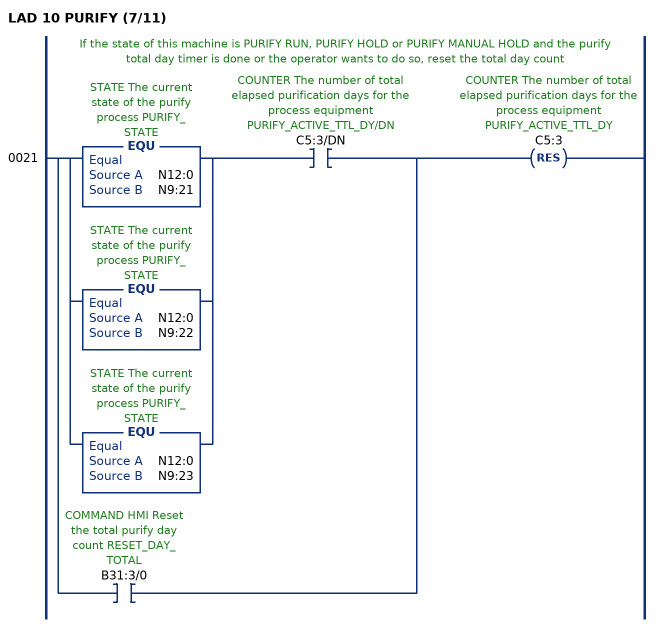
% Rung: 21 %
% If the state of this machine is PURIFY RUN, PURIFY HOLD or PURIFY MANUAL HOLD and the purify total day timer is done or the operator wants to do so, reset the total day count %
SOR BST BST EQU N12:0 N9:21 NXB EQU N12:0 N9:22 NXB EQU N12:0 N9:23 BND XIC C5:3/DN NXB XIC B31:3/0 BND RES C5:3 EOR
%   N12:0  PURIFY_STATE  "STATE The current state of the purify process" %
%   N9:21  PURIFY_RUN  "STATE Purify running" %
%   N9:22  PURIFY_HOLD  "STATE Purify Hold" %
%   N9:23  PURIFY_MANUAL_HOLD  "STATE Purify Manual Hold" %
%   C5:3  PURIFY_ACTIVE_TTL_DY  "COUNTER The number of total elapsed purification days for the process equipment" %
%   B31:3/0  RESET_DAY_TOTAL  "COMMAND HMI Reset the total purify day count" %

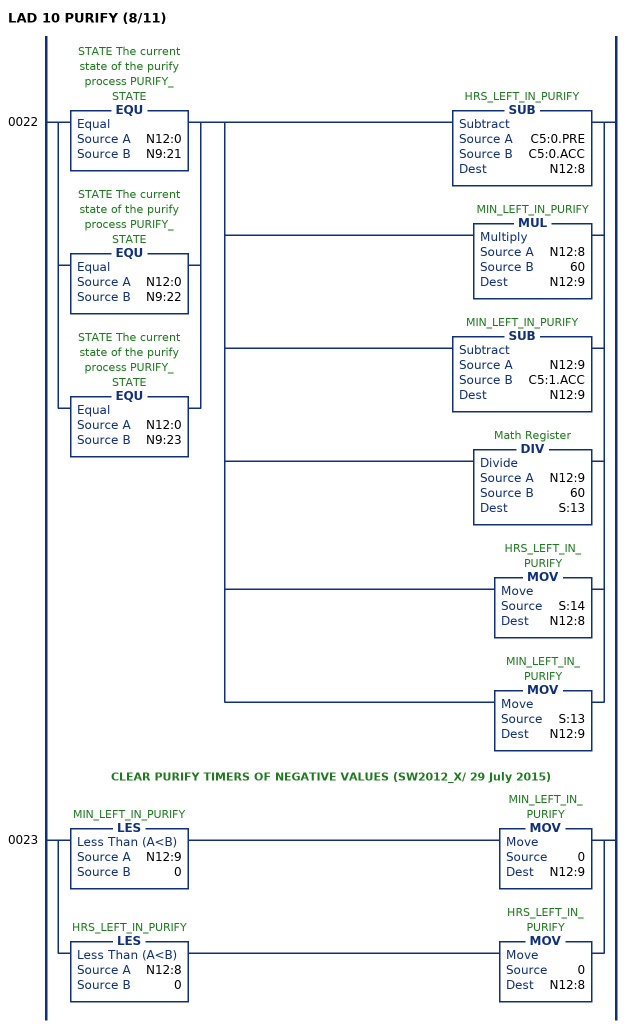
% Rung: 22 %
SOR BST EQU N12:0 N9:21 NXB EQU N12:0 N9:22 NXB EQU N12:0 N9:23 BND BST SUB C5:0.PRE C5:0.ACC N12:8 NXB MUL N12:8 60 N12:9 NXB SUB N12:9 C5:1.ACC N12:9 NXB DIV N12:9 60 S:13 NXB MOV S:14 N12:8 NXB MOV S:13 N12:9 BND EOR
%   N12:0  PURIFY_STATE  "STATE The current state of the purify process" %
%   N9:21  PURIFY_RUN  "STATE Purify running" %
%   N9:22  PURIFY_HOLD  "STATE Purify Hold" %
%   N9:23  PURIFY_MANUAL_HOLD  "STATE Purify Manual Hold" %
%   C5:0  PURIFY_ACTIVE_HOURS  "COUNTER The number of elapsed purification hours for the current ADS" %
%   N12:8  HRS_LEFT_IN_PURIFY %
%   N12:9  MIN_LEFT_IN_PURIFY %
%   C5:1  PURIFY_ACTIVE_MINUTE  "COUNTER The number of elapsed purification minutes for the current ADS (60 min)" %
%   S:13  "Math Register" %
%   S:14  "Math Register" %
% Rung: 23 %
% TITLE: CLEAR PURIFY TIMERS OF NEGATIVE VALUES (SW2012_X/ 29 July 2015) %
SOR BST LES N12:9 0 MOV 0 N12:9 NXB LES N12:8 0 MOV 0 N12:8 BND EOR
%   N12:9  MIN_LEFT_IN_PURIFY %
%   N12:8  HRS_LEFT_IN_PURIFY %

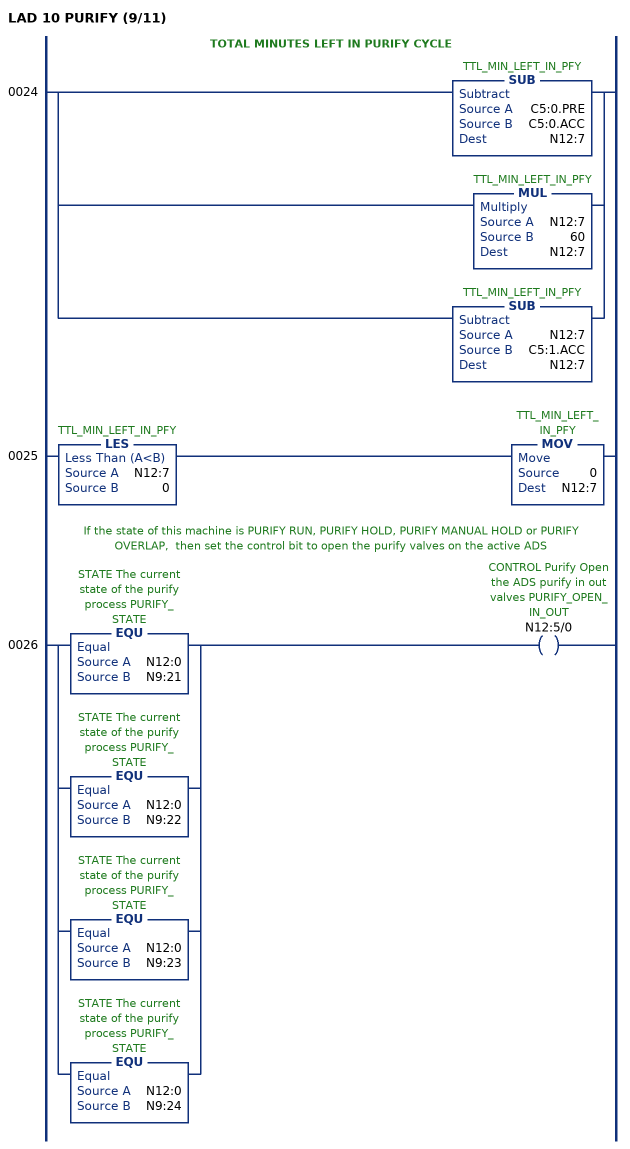
% Rung: 24 %
% TITLE: TOTAL MINUTES LEFT IN PURIFY CYCLE %
SOR BST SUB C5:0.PRE C5:0.ACC N12:7 NXB MUL N12:7 60 N12:7 NXB SUB N12:7 C5:1.ACC N12:7 BND EOR
%   C5:0  PURIFY_ACTIVE_HOURS  "COUNTER The number of elapsed purification hours for the current ADS" %
%   N12:7  TTL_MIN_LEFT_IN_PFY %
%   C5:1  PURIFY_ACTIVE_MINUTE  "COUNTER The number of elapsed purification minutes for the current ADS (60 min)" %
% Rung: 25 %
SOR LES N12:7 0 MOV 0 N12:7 EOR
%   N12:7  TTL_MIN_LEFT_IN_PFY %
% Rung: 26 %
% If the state of this machine is PURIFY RUN, PURIFY HOLD, PURIFY MANUAL HOLD or PURIFY OVERLAP,  then set the control bit to open the purify valves on the active ADS %
SOR BST EQU N12:0 N9:21 NXB EQU N12:0 N9:22 NXB EQU N12:0 N9:23 NXB EQU N12:0 N9:24 BND OTE N12:5/0 EOR
%   N12:0  PURIFY_STATE  "STATE The current state of the purify process" %
%   N9:21  PURIFY_RUN  "STATE Purify running" %
%   N9:22  PURIFY_HOLD  "STATE Purify Hold" %
%   N9:23  PURIFY_MANUAL_HOLD  "STATE Purify Manual Hold" %
%   N9:24  PURIFY_OVERLAP  "STATE Puriify Overlap" %
%   N12:5/0  PURIFY_OPEN_IN_OUT  "CONTROL Purify Open the ADS purify in out valves" %

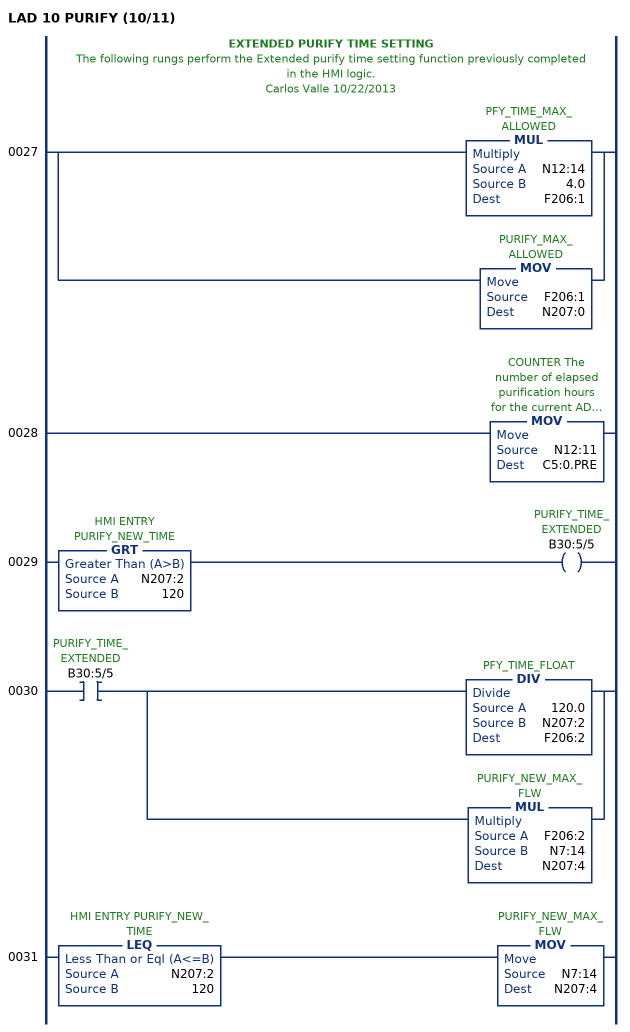
% Rung: 27 %
% TITLE: EXTENDED PURIFY TIME SETTING %
% The following rungs perform the Extended purify time setting function previously completed in the HMI logic.
% Carlos Valle 10/22/2013 %
SOR BST MUL N12:14 4.0 F206:1 NXB MOV F206:1 N207:0 BND EOR
%   N12:14  DEFAULT_PURIFY_TIME %
%   F206:1  PFY_TIME_MAX_ALLOWED %
%   N207:0  PURIFY_MAX_ALLOWED %
% Rung: 28 %
SOR MOV N12:11 C5:0.PRE EOR
%   N12:11  PURIFY_TIME  "CONFIG The time for which the purify operation will occur (hours)" %
%   C5:0  PURIFY_ACTIVE_HOURS  "COUNTER The number of elapsed purification hours for the current ADS" %
% Rung: 29 %
SOR GRT N207:2 120 OTE B30:5/5 EOR
%   N207:2  PURIFY_NEW_TIME  "HMI ENTRY" %
%   B30:5/5  PURIFY_TIME_EXTENDED %
% Rung: 30 %
SOR XIC B30:5/5 BST DIV 120.0 N207:2 F206:2 NXB MUL F206:2 N7:14 N207:4 BND EOR
%   B30:5/5  PURIFY_TIME_EXTENDED %
%   N207:2  PURIFY_NEW_TIME  "HMI ENTRY" %
%   F206:2  PFY_TIME_FLOAT %
%   N7:14  PURIFIER_SIZE %
%   N207:4  PURIFY_NEW_MAX_FLW %
% Rung: 31 %
SOR LEQ N207:2 120 MOV N7:14 N207:4 EOR
%   N207:2  PURIFY_NEW_TIME  "HMI ENTRY" %
%   N7:14  PURIFIER_SIZE %
%   N207:4  PURIFY_NEW_MAX_FLW %

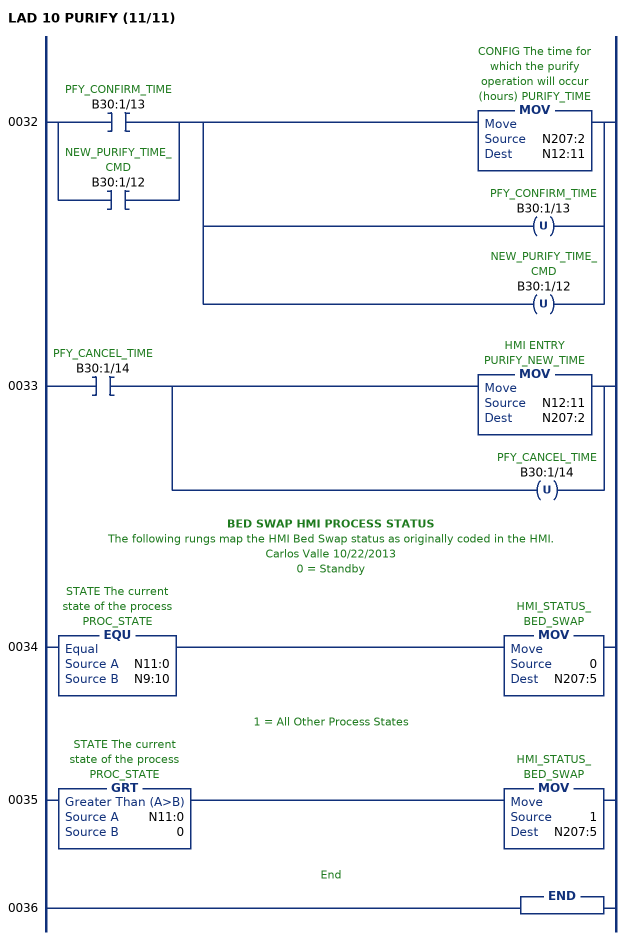
% Rung: 32 %
SOR BST XIC B30:1/13 NXB XIC B30:1/12 BND BST MOV N207:2 N12:11 NXB OTU B30:1/13 NXB OTU B30:1/12 BND EOR
%   B30:1/13  PFY_CONFIRM_TIME %
%   B30:1/12  NEW_PURIFY_TIME_CMD %
%   N207:2  PURIFY_NEW_TIME  "HMI ENTRY" %
%   N12:11  PURIFY_TIME  "CONFIG The time for which the purify operation will occur (hours)" %
% Rung: 33 %
SOR XIC B30:1/14 BST MOV N12:11 N207:2 NXB OTU B30:1/14 BND EOR
%   B30:1/14  PFY_CANCEL_TIME %
%   N12:11  PURIFY_TIME  "CONFIG The time for which the purify operation will occur (hours)" %
%   N207:2  PURIFY_NEW_TIME  "HMI ENTRY" %
% Rung: 34 %
% TITLE: BED SWAP HMI PROCESS STATUS %
% The following rungs map the HMI Bed Swap status as originally coded in the HMI.
% Carlos Valle 10/22/2013
% 0 = Standby %
SOR EQU N11:0 N9:10 MOV 0 N207:5 EOR
%   N11:0  PROC_STATE  "STATE The current state of the process" %
%   N9:10  PROC_STANDBY  "STATE Process Standby" %
%   N207:5  HMI_STATUS_BED_SWAP %
% Rung: 35 %
% 1 = All Other Process States %
SOR GRT N11:0 0 MOV 1 N207:5 EOR
%   N11:0  PROC_STATE  "STATE The current state of the process" %
%   N207:5  HMI_STATUS_BED_SWAP %
% Rung: 36 %
% End %
SOR END EOR

LADDER 11 "REGEN"    % Operates the regen control %
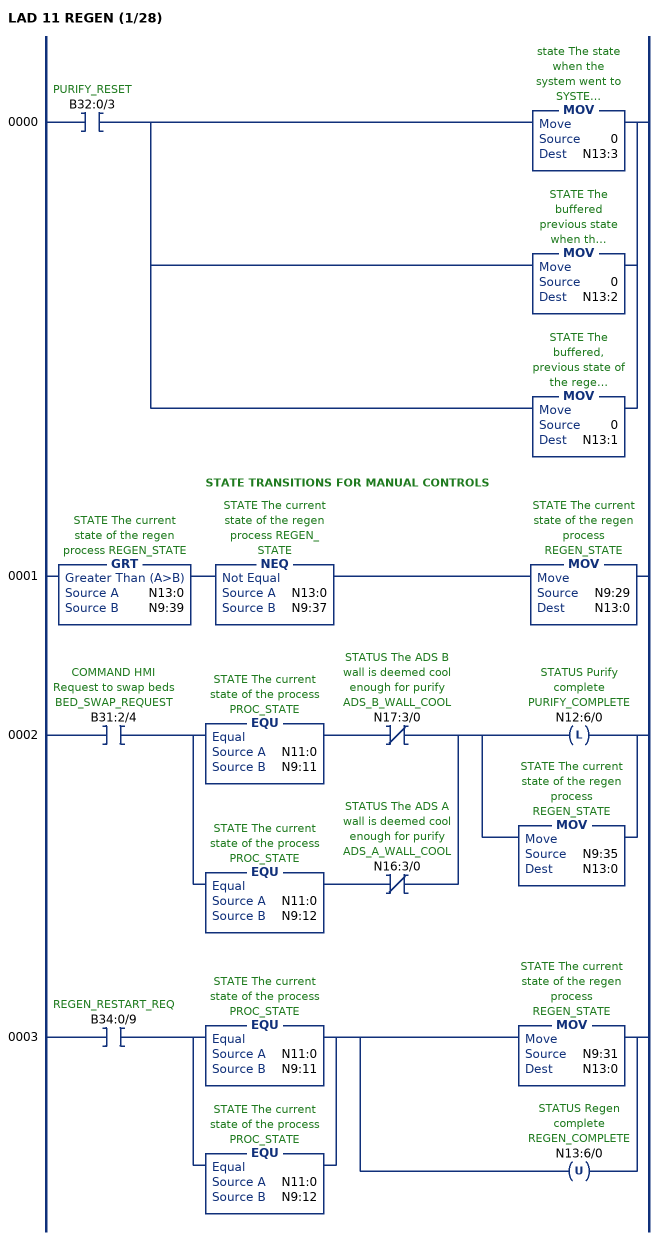
% Rung: 0 %
SOR XIC B32:0/3 BST MOV 0 N13:3 NXB MOV 0 N13:2 NXB MOV 0 N13:1 BND EOR
%   B32:0/3  PURIFY_RESET %
%   N13:3  REGEN_STANDBY_BUFFER  "state The state when the system went to SYSTEM STANDBY" %
%   N13:2  REGEN_ALARM_BUFFER  "STATE The buffered previous state when the system alarm occured" %
%   N13:1  REGEN_BUFFER  "STATE The buffered, previous state of the regen process" %
% Rung: 1 %
% TITLE: STATE TRANSITIONS FOR MANUAL CONTROLS %
SOR GRT N13:0 N9:39 NEQ N13:0 N9:37 MOV N9:29 N13:0 EOR
%   N13:0  REGEN_STATE  "STATE The current state of the regen process" %
%   N9:39  REGEN_EQUALIZE %
%   N9:37  REGEN_ALARM  "STATE Regen Alarm" %
%   N9:29  REGEN_IDLE %
% Rung: 2 %
SOR XIC B31:2/4 BST EQU N11:0 N9:11 XIO N17:3/0 NXB EQU N11:0 N9:12 XIO N16:3/0 BND BST OTL N12:6/0 NXB MOV N9:35 N13:0 BND EOR
%   B31:2/4  BED_SWAP_REQUEST  "COMMAND HMI Request to swap beds" %
%   N11:0  PROC_STATE  "STATE The current state of the process" %
%   N9:11  PROC_PURIFY_A  "STATE Process Purify A" %
%   N17:3/0  ADS_B_WALL_COOL  "STATUS The ADS B wall is deemed cool enough for purify" %
%   N9:12  PROC_PURIFY_B  "STATE Process Purify B" %
%   N16:3/0  ADS_A_WALL_COOL  "STATUS The ADS A wall is deemed cool enough for purify" %
%   N12:6/0  PURIFY_COMPLETE  "STATUS Purify complete" %
%   N9:35  REGEN_COOL_WALL  "STATE Regen Cool wall" %
%   N13:0  REGEN_STATE  "STATE The current state of the regen process" %
% Rung: 3 %
SOR XIC B34:0/9 BST EQU N11:0 N9:11 NXB EQU N11:0 N9:12 BND BST MOV N9:31 N13:0 NXB OTU N13:6/0 BND EOR
%   B34:0/9  REGEN_RESTART_REQ %
%   N11:0  PROC_STATE  "STATE The current state of the process" %
%   N9:11  PROC_PURIFY_A  "STATE Process Purify A" %
%   N9:12  PROC_PURIFY_B  "STATE Process Purify B" %
%   N9:31  REGEN_DELAY  "STATE Regen Delay" %
%   N13:0  REGEN_STATE  "STATE The current state of the regen process" %
%   N13:6/0  REGEN_COMPLETE  "STATUS Regen complete" %

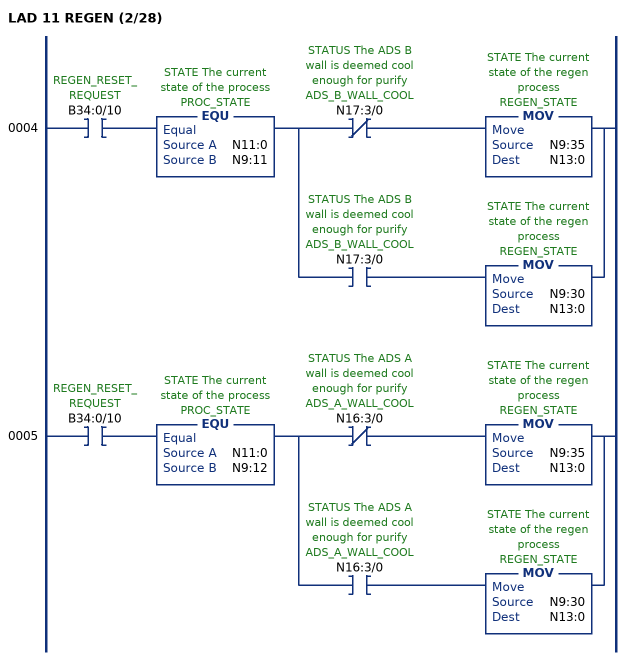
% Rung: 4 %
SOR XIC B34:0/10 EQU N11:0 N9:11 BST XIO N17:3/0 MOV N9:35 N13:0 NXB XIC N17:3/0 MOV N9:30 N13:0 BND EOR
%   B34:0/10  REGEN_RESET_REQUEST %
%   N11:0  PROC_STATE  "STATE The current state of the process" %
%   N9:11  PROC_PURIFY_A  "STATE Process Purify A" %
%   N17:3/0  ADS_B_WALL_COOL  "STATUS The ADS B wall is deemed cool enough for purify" %
%   N9:35  REGEN_COOL_WALL  "STATE Regen Cool wall" %
%   N13:0  REGEN_STATE  "STATE The current state of the regen process" %
%   N9:30  REGEN_STANDBY  "STATE Regen Standby" %
% Rung: 5 %
SOR XIC B34:0/10 EQU N11:0 N9:12 BST XIO N16:3/0 MOV N9:35 N13:0 NXB XIC N16:3/0 MOV N9:30 N13:0 BND EOR
%   B34:0/10  REGEN_RESET_REQUEST %
%   N11:0  PROC_STATE  "STATE The current state of the process" %
%   N9:12  PROC_PURIFY_B  "STATE Process Purify B" %
%   N16:3/0  ADS_A_WALL_COOL  "STATUS The ADS A wall is deemed cool enough for purify" %
%   N9:35  REGEN_COOL_WALL  "STATE Regen Cool wall" %
%   N13:0  REGEN_STATE  "STATE The current state of the regen process" %
%   N9:30  REGEN_STANDBY  "STATE Regen Standby" %

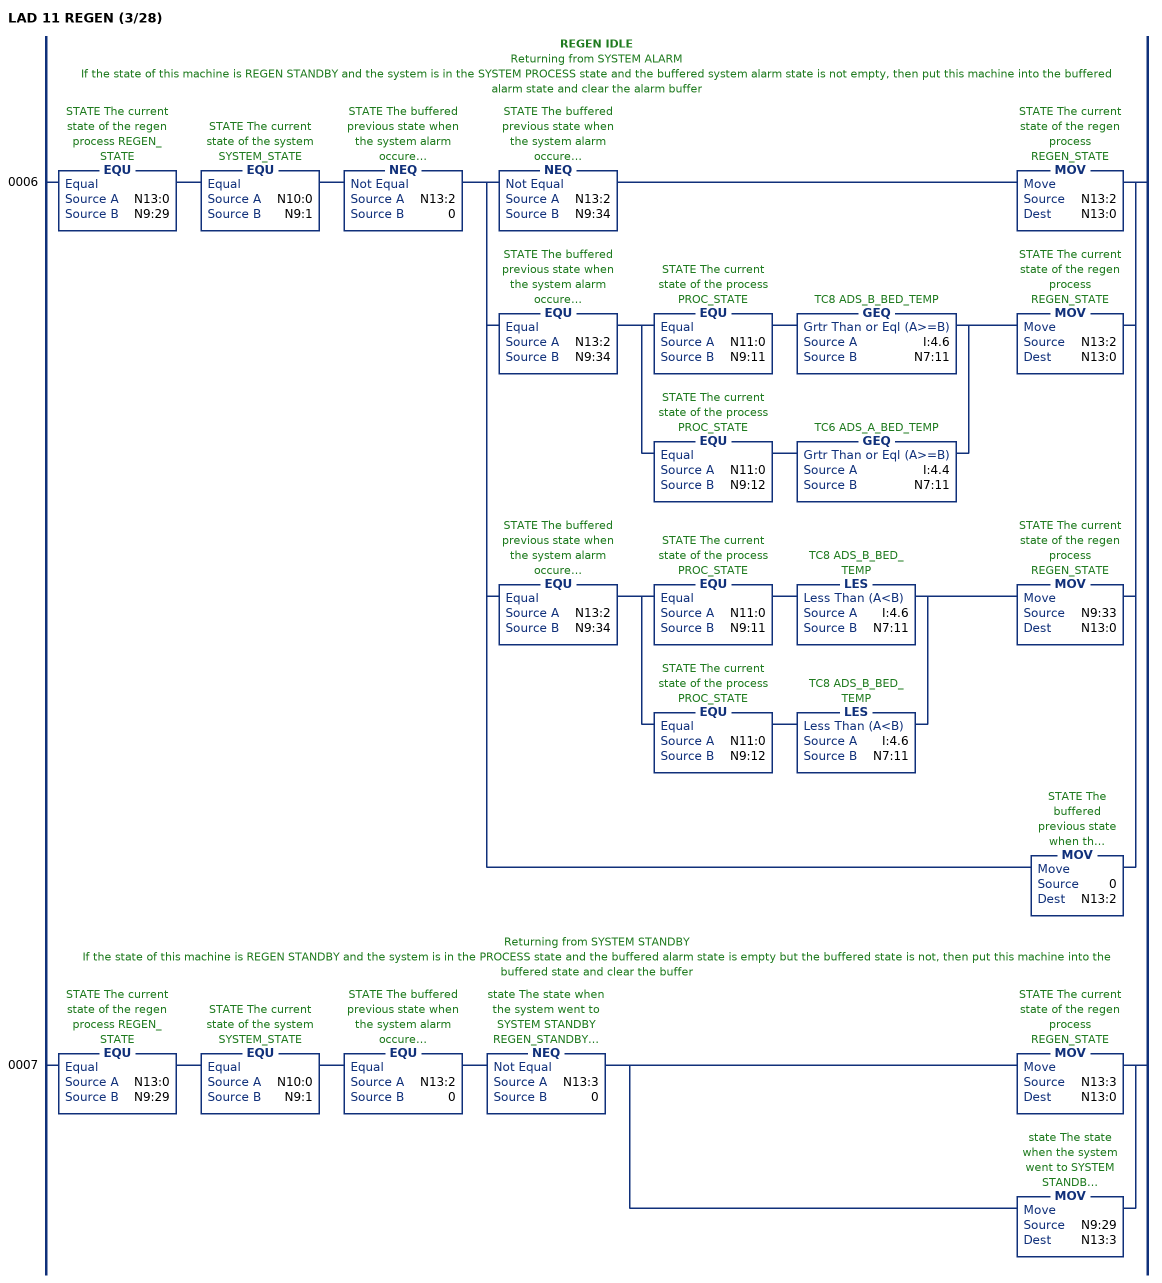
% Rung: 6 %
% TITLE: REGEN IDLE %
% Returning from SYSTEM ALARM
% If the state of this machine is REGEN STANDBY and the system is in the SYSTEM PROCESS state and the buffered system alarm state is not empty, then put this machine into the buffered alarm state and clear the alarm buffer %
SOR EQU N13:0 N9:29 EQU N10:0 N9:1 NEQ N13:2 0 BST NEQ N13:2 N9:34 MOV N13:2 N13:0 NXB EQU N13:2 N9:34 BST EQU N11:0 N9:11 GEQ I:4.6 N7:11 NXB EQU N11:0 N9:12 GEQ I:4.4 N7:11 BND MOV N13:2 N13:0 NXB EQU N13:2 N9:34 BST EQU N11:0 N9:11 LES I:4.6 N7:11 NXB EQU N11:0 N9:12 LES I:4.6 N7:11 BND MOV N9:33 N13:0 NXB MOV 0 N13:2 BND EOR
%   N13:0  REGEN_STATE  "STATE The current state of the regen process" %
%   N9:29  REGEN_IDLE %
%   N10:0  SYSTEM_STATE  "STATE The current state of the system" %
%   N9:1  SYSTEM_PROCESS  "STATE System Process" %
%   N13:2  REGEN_ALARM_BUFFER  "STATE The buffered previous state when the system alarm occured" %
%   N9:34  REGEN_H2_REDUCTION  "STATE Regen Running" %
%   N11:0  PROC_STATE  "STATE The current state of the process" %
%   N9:11  PROC_PURIFY_A  "STATE Process Purify A" %
%   I:4.6  ADS_B_BED_TEMP  "TC8" %
%   N7:11  ADS_BED_TEMP_HIGH  "CONFIG The temp at which the regen process may continue" %
%   N9:12  PROC_PURIFY_B  "STATE Process Purify B" %
%   I:4.4  ADS_A_BED_TEMP  "TC6" %
%   N9:33  REGEN_HEAT_BED  "STATE Regen Heat wall" %
% Rung: 7 %
% Returning from SYSTEM STANDBY
% If the state of this machine is REGEN STANDBY and the system is in the PROCESS state and the buffered alarm state is empty but the buffered state is not, then put this machine into the buffered state and clear the buffer %
SOR EQU N13:0 N9:29 EQU N10:0 N9:1 EQU N13:2 0 NEQ N13:3 0 BST MOV N13:3 N13:0 NXB MOV N9:29 N13:3 BND EOR
%   N13:0  REGEN_STATE  "STATE The current state of the regen process" %
%   N9:29  REGEN_IDLE %
%   N10:0  SYSTEM_STATE  "STATE The current state of the system" %
%   N9:1  SYSTEM_PROCESS  "STATE System Process" %
%   N13:2  REGEN_ALARM_BUFFER  "STATE The buffered previous state when the system alarm occured" %
%   N13:3  REGEN_STANDBY_BUFFER  "state The state when the system went to SYSTEM STANDBY" %

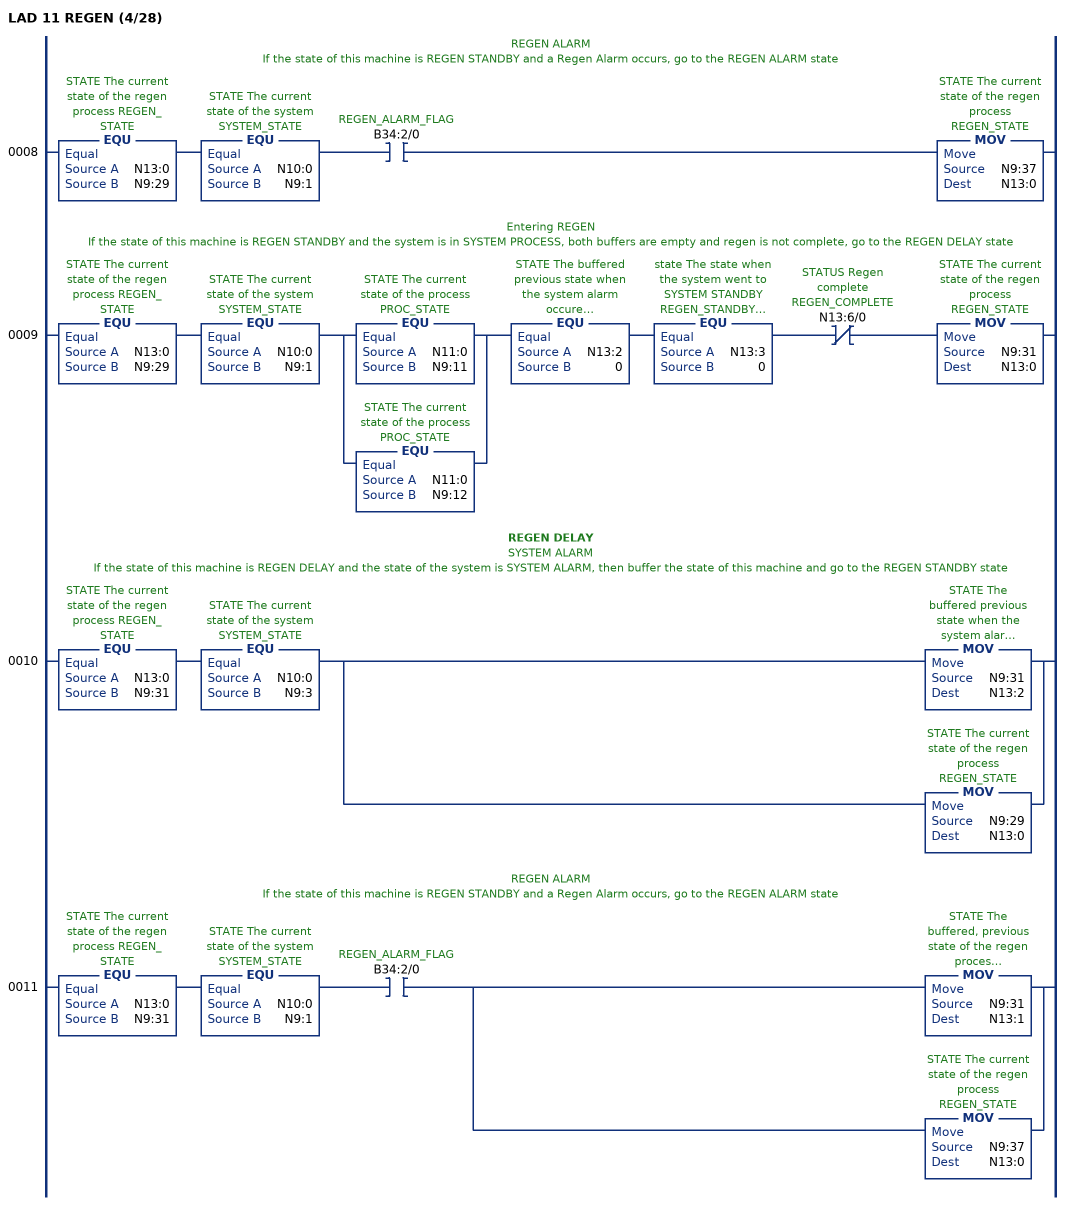
% Rung: 8 %
% REGEN ALARM
% If the state of this machine is REGEN STANDBY and a Regen Alarm occurs, go to the REGEN ALARM state %
SOR EQU N13:0 N9:29 EQU N10:0 N9:1 XIC B34:2/0 MOV N9:37 N13:0 EOR
%   N13:0  REGEN_STATE  "STATE The current state of the regen process" %
%   N9:29  REGEN_IDLE %
%   N10:0  SYSTEM_STATE  "STATE The current state of the system" %
%   N9:1  SYSTEM_PROCESS  "STATE System Process" %
%   B34:2/0  REGEN_ALARM_FLAG %
%   N9:37  REGEN_ALARM  "STATE Regen Alarm" %
% Rung: 9 %
% Entering REGEN
% If the state of this machine is REGEN STANDBY and the system is in SYSTEM PROCESS, both buffers are empty and regen is not complete, go to the REGEN DELAY state %
SOR EQU N13:0 N9:29 EQU N10:0 N9:1 BST EQU N11:0 N9:11 NXB EQU N11:0 N9:12 BND EQU N13:2 0 EQU N13:3 0 XIO N13:6/0 MOV N9:31 N13:0 EOR
%   N13:0  REGEN_STATE  "STATE The current state of the regen process" %
%   N9:29  REGEN_IDLE %
%   N10:0  SYSTEM_STATE  "STATE The current state of the system" %
%   N9:1  SYSTEM_PROCESS  "STATE System Process" %
%   N11:0  PROC_STATE  "STATE The current state of the process" %
%   N9:11  PROC_PURIFY_A  "STATE Process Purify A" %
%   N9:12  PROC_PURIFY_B  "STATE Process Purify B" %
%   N13:2  REGEN_ALARM_BUFFER  "STATE The buffered previous state when the system alarm occured" %
%   N13:3  REGEN_STANDBY_BUFFER  "state The state when the system went to SYSTEM STANDBY" %
%   N13:6/0  REGEN_COMPLETE  "STATUS Regen complete" %
%   N9:31  REGEN_DELAY  "STATE Regen Delay" %
% Rung: 10 %
% TITLE: REGEN DELAY %
% SYSTEM ALARM
% If the state of this machine is REGEN DELAY and the state of the system is SYSTEM ALARM, then buffer the state of this machine and go to the REGEN STANDBY state %
SOR EQU N13:0 N9:31 EQU N10:0 N9:3 BST MOV N9:31 N13:2 NXB MOV N9:29 N13:0 BND EOR
%   N13:0  REGEN_STATE  "STATE The current state of the regen process" %
%   N9:31  REGEN_DELAY  "STATE Regen Delay" %
%   N10:0  SYSTEM_STATE  "STATE The current state of the system" %
%   N9:3  SYSTEM_ALARM  "STATE System Alarm" %
%   N13:2  REGEN_ALARM_BUFFER  "STATE The buffered previous state when the system alarm occured" %
%   N9:29  REGEN_IDLE %
% Rung: 11 %
% REGEN ALARM
% If the state of this machine is REGEN STANDBY and a Regen Alarm occurs, go to the REGEN ALARM state %
SOR EQU N13:0 N9:31 EQU N10:0 N9:1 XIC B34:2/0 BST MOV N9:31 N13:1 NXB MOV N9:37 N13:0 BND EOR
%   N13:0  REGEN_STATE  "STATE The current state of the regen process" %
%   N9:31  REGEN_DELAY  "STATE Regen Delay" %
%   N10:0  SYSTEM_STATE  "STATE The current state of the system" %
%   N9:1  SYSTEM_PROCESS  "STATE System Process" %
%   B34:2/0  REGEN_ALARM_FLAG %
%   N13:1  REGEN_BUFFER  "STATE The buffered, previous state of the regen process" %
%   N9:37  REGEN_ALARM  "STATE Regen Alarm" %

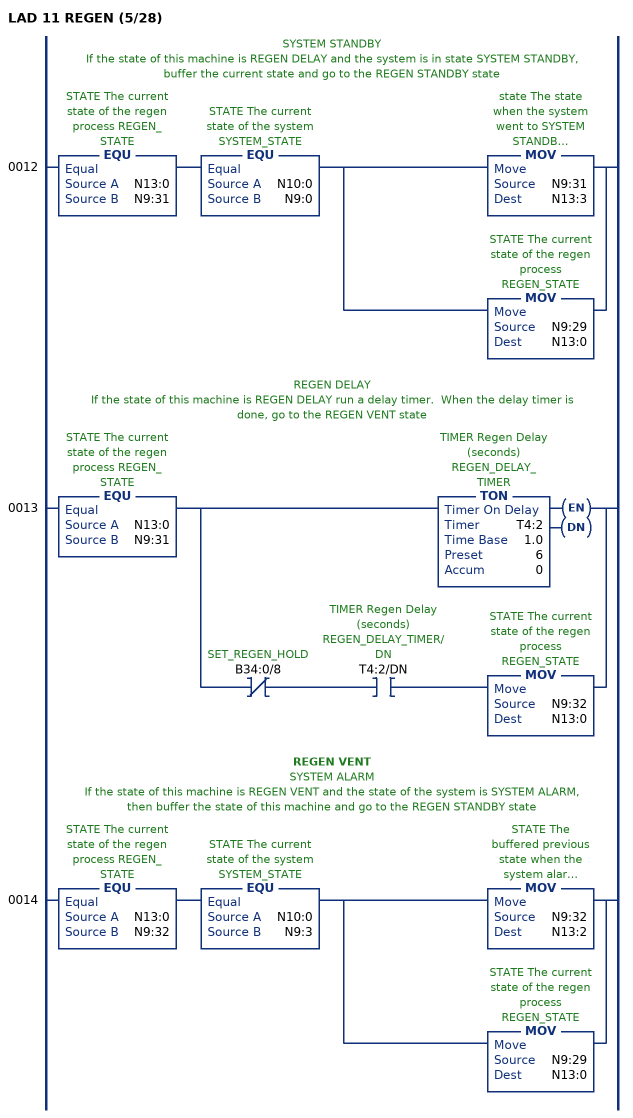
% Rung: 12 %
% SYSTEM STANDBY
% If the state of this machine is REGEN DELAY and the system is in state SYSTEM STANDBY, buffer the current state and go to the REGEN STANDBY state %
SOR EQU N13:0 N9:31 EQU N10:0 N9:0 BST MOV N9:31 N13:3 NXB MOV N9:29 N13:0 BND EOR
%   N13:0  REGEN_STATE  "STATE The current state of the regen process" %
%   N9:31  REGEN_DELAY  "STATE Regen Delay" %
%   N10:0  SYSTEM_STATE  "STATE The current state of the system" %
%   N9:0  SYSTEM_STANDBY  "STATE System Standby" %
%   N13:3  REGEN_STANDBY_BUFFER  "state The state when the system went to SYSTEM STANDBY" %
%   N9:29  REGEN_IDLE %
% Rung: 13 %
% REGEN DELAY
% If the state of this machine is REGEN DELAY run a delay timer.  When the delay timer is done, go to the REGEN VENT state %
SOR EQU N13:0 N9:31 BST TON T4:2 1.0 6 0 NXB XIO B34:0/8 XIC T4:2/DN MOV N9:32 N13:0 BND EOR
%   N13:0  REGEN_STATE  "STATE The current state of the regen process" %
%   N9:31  REGEN_DELAY  "STATE Regen Delay" %
%   T4:2  REGEN_DELAY_TIMER  "TIMER Regen Delay (seconds)" %
%   B34:0/8  SET_REGEN_HOLD %
%   N9:32  REGEN_VENT  "STATE Regen Vent" %
% Rung: 14 %
% TITLE: REGEN VENT %
% SYSTEM ALARM
% If the state of this machine is REGEN VENT and the state of the system is SYSTEM ALARM, then buffer the state of this machine and go to the REGEN STANDBY state %
SOR EQU N13:0 N9:32 EQU N10:0 N9:3 BST MOV N9:32 N13:2 NXB MOV N9:29 N13:0 BND EOR
%   N13:0  REGEN_STATE  "STATE The current state of the regen process" %
%   N9:32  REGEN_VENT  "STATE Regen Vent" %
%   N10:0  SYSTEM_STATE  "STATE The current state of the system" %
%   N9:3  SYSTEM_ALARM  "STATE System Alarm" %
%   N13:2  REGEN_ALARM_BUFFER  "STATE The buffered previous state when the system alarm occured" %
%   N9:29  REGEN_IDLE %

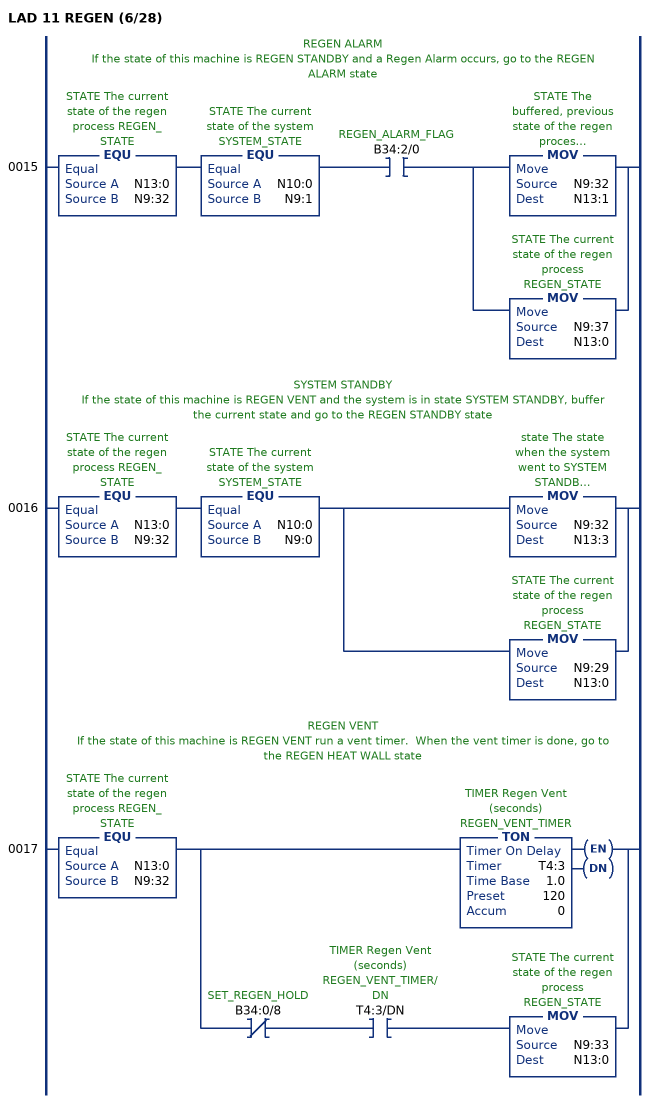
% Rung: 15 %
% REGEN ALARM
% If the state of this machine is REGEN STANDBY and a Regen Alarm occurs, go to the REGEN ALARM state %
SOR EQU N13:0 N9:32 EQU N10:0 N9:1 XIC B34:2/0 BST MOV N9:32 N13:1 NXB MOV N9:37 N13:0 BND EOR
%   N13:0  REGEN_STATE  "STATE The current state of the regen process" %
%   N9:32  REGEN_VENT  "STATE Regen Vent" %
%   N10:0  SYSTEM_STATE  "STATE The current state of the system" %
%   N9:1  SYSTEM_PROCESS  "STATE System Process" %
%   B34:2/0  REGEN_ALARM_FLAG %
%   N13:1  REGEN_BUFFER  "STATE The buffered, previous state of the regen process" %
%   N9:37  REGEN_ALARM  "STATE Regen Alarm" %
% Rung: 16 %
% SYSTEM STANDBY
% If the state of this machine is REGEN VENT and the system is in state SYSTEM STANDBY, buffer the current state and go to the REGEN STANDBY state %
SOR EQU N13:0 N9:32 EQU N10:0 N9:0 BST MOV N9:32 N13:3 NXB MOV N9:29 N13:0 BND EOR
%   N13:0  REGEN_STATE  "STATE The current state of the regen process" %
%   N9:32  REGEN_VENT  "STATE Regen Vent" %
%   N10:0  SYSTEM_STATE  "STATE The current state of the system" %
%   N9:0  SYSTEM_STANDBY  "STATE System Standby" %
%   N13:3  REGEN_STANDBY_BUFFER  "state The state when the system went to SYSTEM STANDBY" %
%   N9:29  REGEN_IDLE %
% Rung: 17 %
% REGEN VENT
% If the state of this machine is REGEN VENT run a vent timer.  When the vent timer is done, go to the REGEN HEAT WALL state %
SOR EQU N13:0 N9:32 BST TON T4:3 1.0 120 0 NXB XIO B34:0/8 XIC T4:3/DN MOV N9:33 N13:0 BND EOR
%   N13:0  REGEN_STATE  "STATE The current state of the regen process" %
%   N9:32  REGEN_VENT  "STATE Regen Vent" %
%   T4:3  REGEN_VENT_TIMER  "TIMER Regen Vent (seconds)" %
%   B34:0/8  SET_REGEN_HOLD %
%   N9:33  REGEN_HEAT_BED  "STATE Regen Heat wall" %

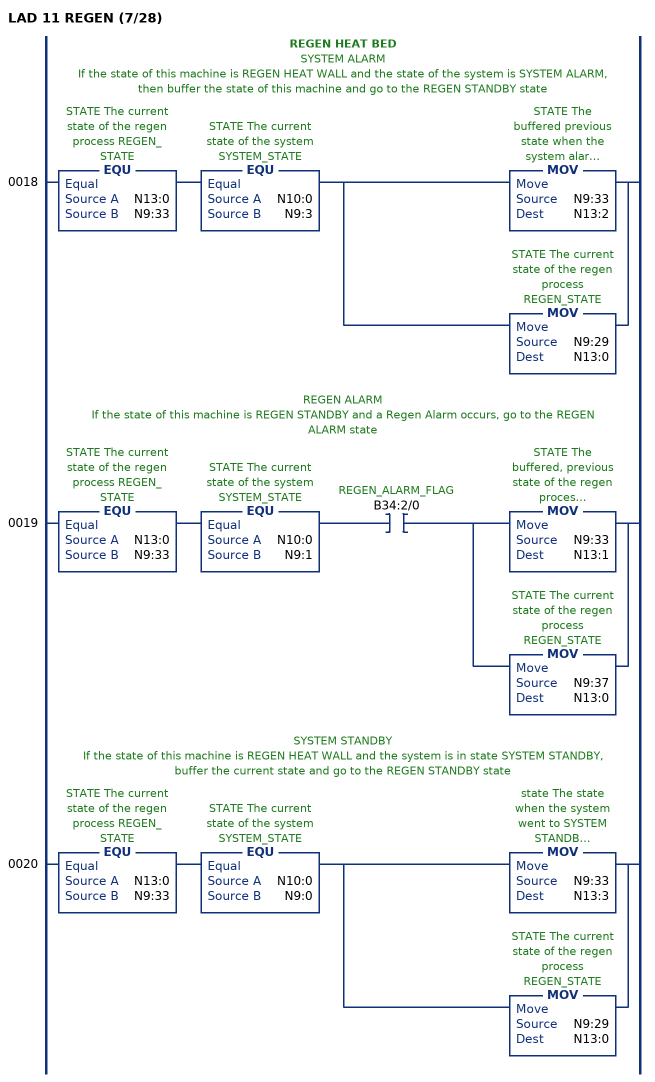
% Rung: 18 %
% TITLE: REGEN HEAT BED %
% SYSTEM ALARM
% If the state of this machine is REGEN HEAT WALL and the state of the system is SYSTEM ALARM, then buffer the state of this machine and go to the REGEN STANDBY state %
SOR EQU N13:0 N9:33 EQU N10:0 N9:3 BST MOV N9:33 N13:2 NXB MOV N9:29 N13:0 BND EOR
%   N13:0  REGEN_STATE  "STATE The current state of the regen process" %
%   N9:33  REGEN_HEAT_BED  "STATE Regen Heat wall" %
%   N10:0  SYSTEM_STATE  "STATE The current state of the system" %
%   N9:3  SYSTEM_ALARM  "STATE System Alarm" %
%   N13:2  REGEN_ALARM_BUFFER  "STATE The buffered previous state when the system alarm occured" %
%   N9:29  REGEN_IDLE %
% Rung: 19 %
% REGEN ALARM
% If the state of this machine is REGEN STANDBY and a Regen Alarm occurs, go to the REGEN ALARM state %
SOR EQU N13:0 N9:33 EQU N10:0 N9:1 XIC B34:2/0 BST MOV N9:33 N13:1 NXB MOV N9:37 N13:0 BND EOR
%   N13:0  REGEN_STATE  "STATE The current state of the regen process" %
%   N9:33  REGEN_HEAT_BED  "STATE Regen Heat wall" %
%   N10:0  SYSTEM_STATE  "STATE The current state of the system" %
%   N9:1  SYSTEM_PROCESS  "STATE System Process" %
%   B34:2/0  REGEN_ALARM_FLAG %
%   N13:1  REGEN_BUFFER  "STATE The buffered, previous state of the regen process" %
%   N9:37  REGEN_ALARM  "STATE Regen Alarm" %
% Rung: 20 %
% SYSTEM STANDBY
% If the state of this machine is REGEN HEAT WALL and the system is in state SYSTEM STANDBY, buffer the current state and go to the REGEN STANDBY state %
SOR EQU N13:0 N9:33 EQU N10:0 N9:0 BST MOV N9:33 N13:3 NXB MOV N9:29 N13:0 BND EOR
%   N13:0  REGEN_STATE  "STATE The current state of the regen process" %
%   N9:33  REGEN_HEAT_BED  "STATE Regen Heat wall" %
%   N10:0  SYSTEM_STATE  "STATE The current state of the system" %
%   N9:0  SYSTEM_STANDBY  "STATE System Standby" %
%   N13:3  REGEN_STANDBY_BUFFER  "state The state when the system went to SYSTEM STANDBY" %
%   N9:29  REGEN_IDLE %

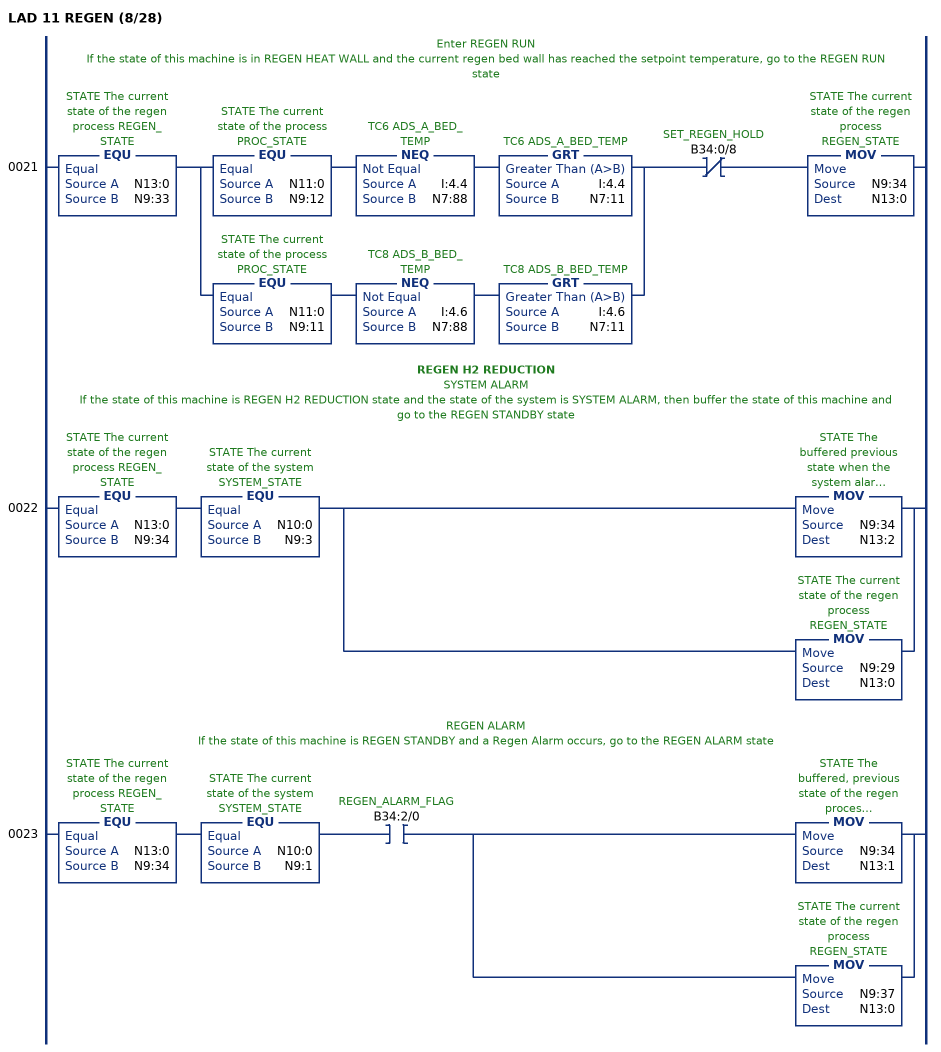
% Rung: 21 %
% Enter REGEN RUN
% If the state of this machine is in REGEN HEAT WALL and the current regen bed wall has reached the setpoint temperature, go to the REGEN RUN state %
SOR EQU N13:0 N9:33 BST EQU N11:0 N9:12 NEQ I:4.4 N7:88 GRT I:4.4 N7:11 NXB EQU N11:0 N9:11 NEQ I:4.6 N7:88 GRT I:4.6 N7:11 BND XIO B34:0/8 MOV N9:34 N13:0 EOR
%   N13:0  REGEN_STATE  "STATE The current state of the regen process" %
%   N9:33  REGEN_HEAT_BED  "STATE Regen Heat wall" %
%   N11:0  PROC_STATE  "STATE The current state of the process" %
%   N9:12  PROC_PURIFY_B  "STATE Process Purify B" %
%   I:4.4  ADS_A_BED_TEMP  "TC6" %
%   N7:88  TC_OPEN_SP  "CONFIG The value read by an open TC input" %
%   N7:11  ADS_BED_TEMP_HIGH  "CONFIG The temp at which the regen process may continue" %
%   N9:11  PROC_PURIFY_A  "STATE Process Purify A" %
%   I:4.6  ADS_B_BED_TEMP  "TC8" %
%   B34:0/8  SET_REGEN_HOLD %
%   N9:34  REGEN_H2_REDUCTION  "STATE Regen Running" %
% Rung: 22 %
% TITLE: REGEN H2 REDUCTION %
% SYSTEM ALARM
% If the state of this machine is REGEN H2 REDUCTION state and the state of the system is SYSTEM ALARM, then buffer the state of this machine and go to the REGEN STANDBY state %
SOR EQU N13:0 N9:34 EQU N10:0 N9:3 BST MOV N9:34 N13:2 NXB MOV N9:29 N13:0 BND EOR
%   N13:0  REGEN_STATE  "STATE The current state of the regen process" %
%   N9:34  REGEN_H2_REDUCTION  "STATE Regen Running" %
%   N10:0  SYSTEM_STATE  "STATE The current state of the system" %
%   N9:3  SYSTEM_ALARM  "STATE System Alarm" %
%   N13:2  REGEN_ALARM_BUFFER  "STATE The buffered previous state when the system alarm occured" %
%   N9:29  REGEN_IDLE %
% Rung: 23 %
% REGEN ALARM
% If the state of this machine is REGEN STANDBY and a Regen Alarm occurs, go to the REGEN ALARM state %
SOR EQU N13:0 N9:34 EQU N10:0 N9:1 XIC B34:2/0 BST MOV N9:34 N13:1 NXB MOV N9:37 N13:0 BND EOR
%   N13:0  REGEN_STATE  "STATE The current state of the regen process" %
%   N9:34  REGEN_H2_REDUCTION  "STATE Regen Running" %
%   N10:0  SYSTEM_STATE  "STATE The current state of the system" %
%   N9:1  SYSTEM_PROCESS  "STATE System Process" %
%   B34:2/0  REGEN_ALARM_FLAG %
%   N13:1  REGEN_BUFFER  "STATE The buffered, previous state of the regen process" %
%   N9:37  REGEN_ALARM  "STATE Regen Alarm" %

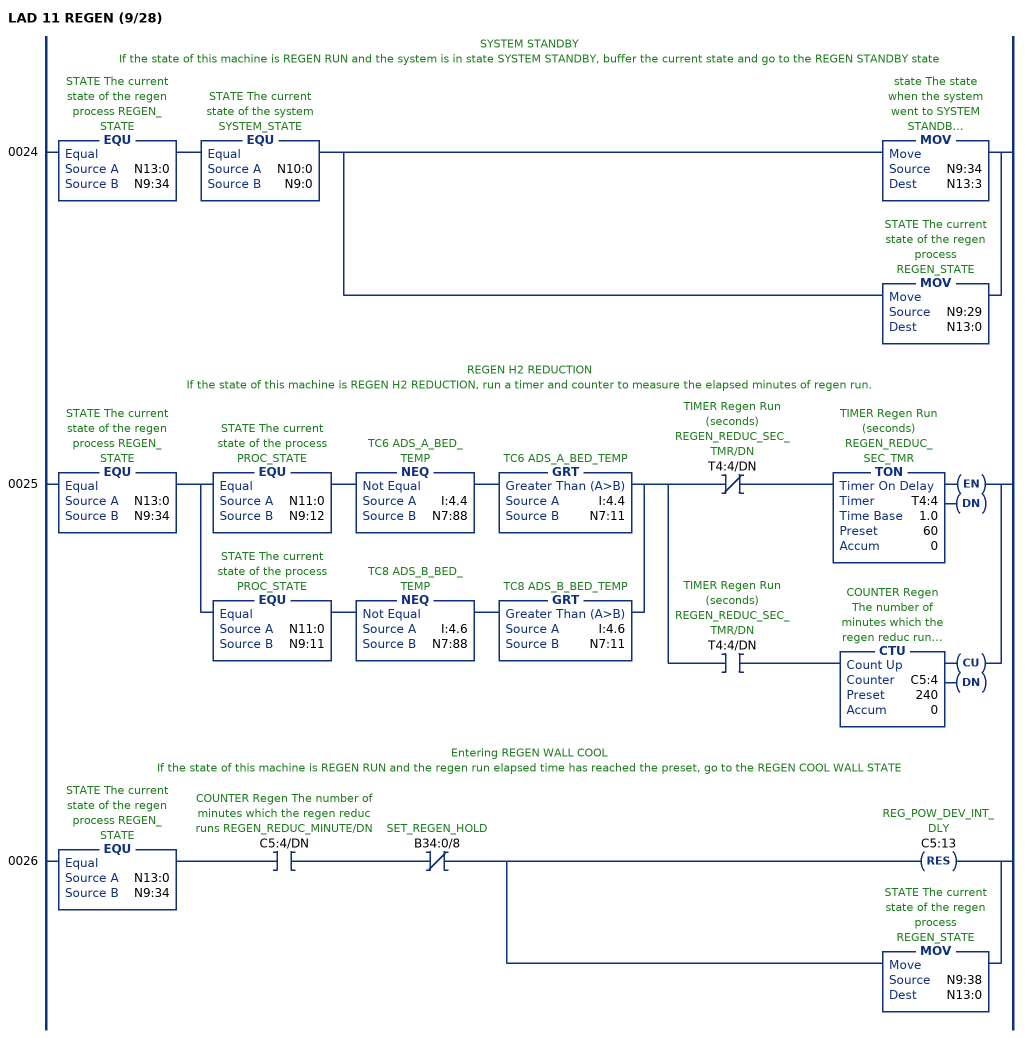
% Rung: 24 %
% SYSTEM STANDBY
% If the state of this machine is REGEN RUN and the system is in state SYSTEM STANDBY, buffer the current state and go to the REGEN STANDBY state %
SOR EQU N13:0 N9:34 EQU N10:0 N9:0 BST MOV N9:34 N13:3 NXB MOV N9:29 N13:0 BND EOR
%   N13:0  REGEN_STATE  "STATE The current state of the regen process" %
%   N9:34  REGEN_H2_REDUCTION  "STATE Regen Running" %
%   N10:0  SYSTEM_STATE  "STATE The current state of the system" %
%   N9:0  SYSTEM_STANDBY  "STATE System Standby" %
%   N13:3  REGEN_STANDBY_BUFFER  "state The state when the system went to SYSTEM STANDBY" %
%   N9:29  REGEN_IDLE %
% Rung: 25 %
% REGEN H2 REDUCTION
% If the state of this machine is REGEN H2 REDUCTION, run a timer and counter to measure the elapsed minutes of regen run. %
SOR EQU N13:0 N9:34 BST EQU N11:0 N9:12 NEQ I:4.4 N7:88 GRT I:4.4 N7:11 NXB EQU N11:0 N9:11 NEQ I:4.6 N7:88 GRT I:4.6 N7:11 BND BST XIO T4:4/DN TON T4:4 1.0 60 0 NXB XIC T4:4/DN CTU C5:4 240 0 BND EOR
%   N13:0  REGEN_STATE  "STATE The current state of the regen process" %
%   N9:34  REGEN_H2_REDUCTION  "STATE Regen Running" %
%   N11:0  PROC_STATE  "STATE The current state of the process" %
%   N9:12  PROC_PURIFY_B  "STATE Process Purify B" %
%   I:4.4  ADS_A_BED_TEMP  "TC6" %
%   N7:88  TC_OPEN_SP  "CONFIG The value read by an open TC input" %
%   N7:11  ADS_BED_TEMP_HIGH  "CONFIG The temp at which the regen process may continue" %
%   N9:11  PROC_PURIFY_A  "STATE Process Purify A" %
%   I:4.6  ADS_B_BED_TEMP  "TC8" %
%   T4:4  REGEN_REDUC_SEC_TMR  "TIMER Regen Run (seconds)" %
%   C5:4  REGEN_REDUC_MINUTE  "COUNTER Regen The number of minutes which the regen reduc runs" %
% Rung: 26 %
% Entering REGEN WALL COOL
% If the state of this machine is REGEN RUN and the regen run elapsed time has reached the preset, go to the REGEN COOL WALL STATE %
SOR EQU N13:0 N9:34 XIC C5:4/DN XIO B34:0/8 BST RES C5:13 NXB MOV N9:38 N13:0 BND EOR
%   N13:0  REGEN_STATE  "STATE The current state of the regen process" %
%   N9:34  REGEN_H2_REDUCTION  "STATE Regen Running" %
%   C5:4  REGEN_REDUC_MINUTE  "COUNTER Regen The number of minutes which the regen reduc runs" %
%   B34:0/8  SET_REGEN_HOLD %
%   C5:13  REG_POW_DEV_INT_DLY %
%   N9:38  REGEN_PURGE  "STATE Regen Hot Purge" %

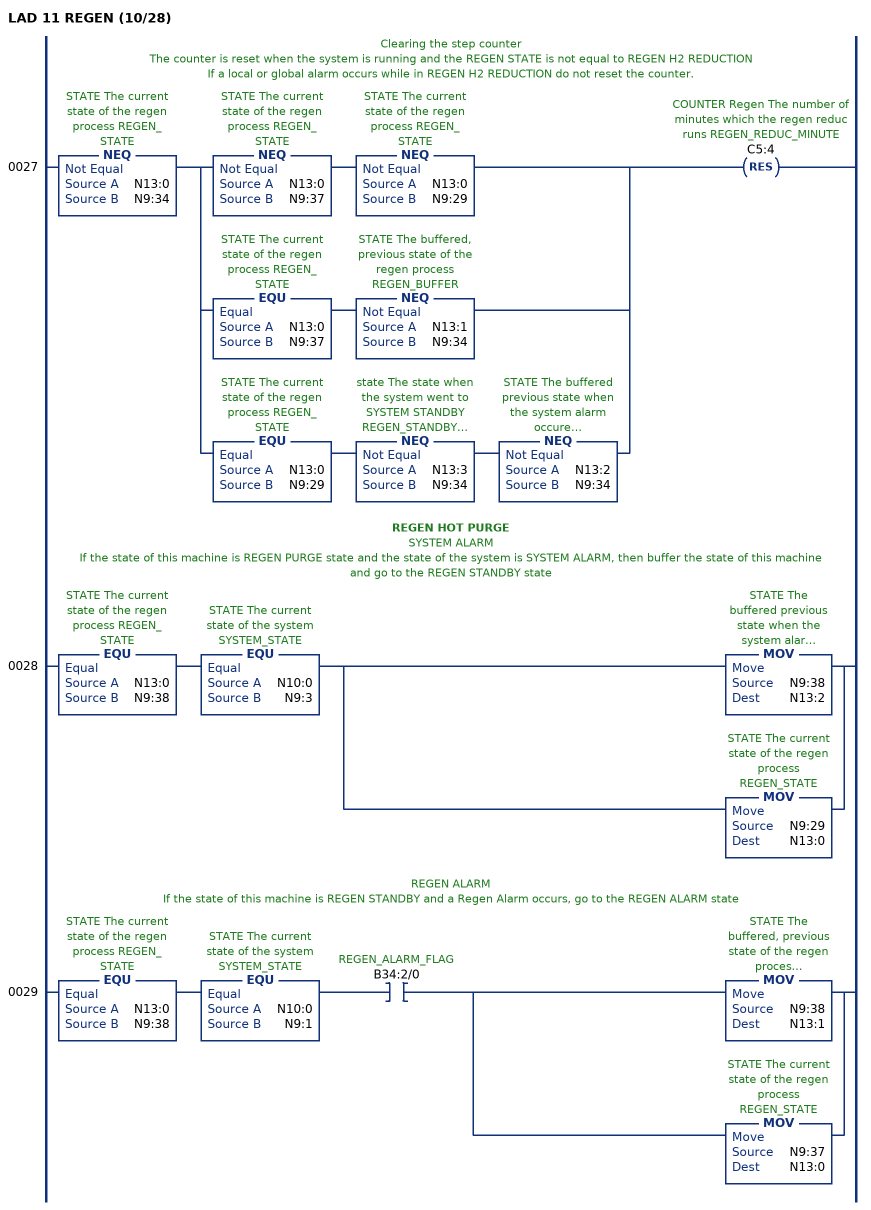
% Rung: 27 %
% Clearing the step counter
% The counter is reset when the system is running and the REGEN STATE is not equal to REGEN H2 REDUCTION
% If a local or global alarm occurs while in REGEN H2 REDUCTION do not reset the counter. %
SOR NEQ N13:0 N9:34 BST NEQ N13:0 N9:37 NEQ N13:0 N9:29 NXB EQU N13:0 N9:37 NEQ N13:1 N9:34 NXB EQU N13:0 N9:29 NEQ N13:3 N9:34 NEQ N13:2 N9:34 BND RES C5:4 EOR
%   N13:0  REGEN_STATE  "STATE The current state of the regen process" %
%   N9:34  REGEN_H2_REDUCTION  "STATE Regen Running" %
%   N9:37  REGEN_ALARM  "STATE Regen Alarm" %
%   N9:29  REGEN_IDLE %
%   N13:1  REGEN_BUFFER  "STATE The buffered, previous state of the regen process" %
%   N13:3  REGEN_STANDBY_BUFFER  "state The state when the system went to SYSTEM STANDBY" %
%   N13:2  REGEN_ALARM_BUFFER  "STATE The buffered previous state when the system alarm occured" %
%   C5:4  REGEN_REDUC_MINUTE  "COUNTER Regen The number of minutes which the regen reduc runs" %
% Rung: 28 %
% TITLE: REGEN HOT PURGE %
% SYSTEM ALARM
% If the state of this machine is REGEN PURGE state and the state of the system is SYSTEM ALARM, then buffer the state of this machine and go to the REGEN STANDBY state %
SOR EQU N13:0 N9:38 EQU N10:0 N9:3 BST MOV N9:38 N13:2 NXB MOV N9:29 N13:0 BND EOR
%   N13:0  REGEN_STATE  "STATE The current state of the regen process" %
%   N9:38  REGEN_PURGE  "STATE Regen Hot Purge" %
%   N10:0  SYSTEM_STATE  "STATE The current state of the system" %
%   N9:3  SYSTEM_ALARM  "STATE System Alarm" %
%   N13:2  REGEN_ALARM_BUFFER  "STATE The buffered previous state when the system alarm occured" %
%   N9:29  REGEN_IDLE %
% Rung: 29 %
% REGEN ALARM
% If the state of this machine is REGEN STANDBY and a Regen Alarm occurs, go to the REGEN ALARM state %
SOR EQU N13:0 N9:38 EQU N10:0 N9:1 XIC B34:2/0 BST MOV N9:38 N13:1 NXB MOV N9:37 N13:0 BND EOR
%   N13:0  REGEN_STATE  "STATE The current state of the regen process" %
%   N9:38  REGEN_PURGE  "STATE Regen Hot Purge" %
%   N10:0  SYSTEM_STATE  "STATE The current state of the system" %
%   N9:1  SYSTEM_PROCESS  "STATE System Process" %
%   B34:2/0  REGEN_ALARM_FLAG %
%   N13:1  REGEN_BUFFER  "STATE The buffered, previous state of the regen process" %
%   N9:37  REGEN_ALARM  "STATE Regen Alarm" %

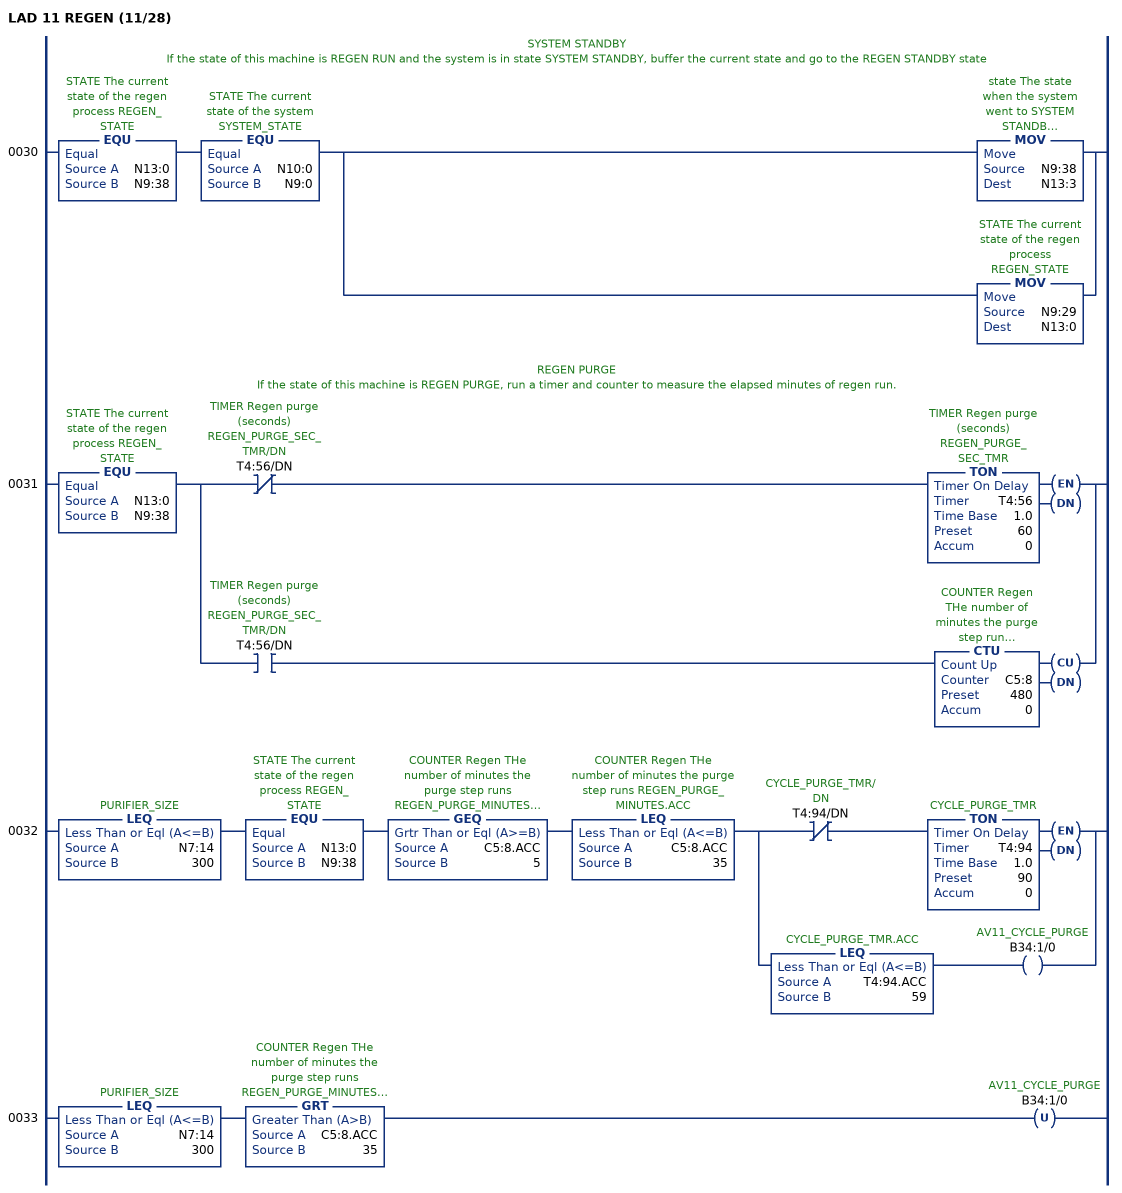
% Rung: 30 %
% SYSTEM STANDBY
% If the state of this machine is REGEN RUN and the system is in state SYSTEM STANDBY, buffer the current state and go to the REGEN STANDBY state %
SOR EQU N13:0 N9:38 EQU N10:0 N9:0 BST MOV N9:38 N13:3 NXB MOV N9:29 N13:0 BND EOR
%   N13:0  REGEN_STATE  "STATE The current state of the regen process" %
%   N9:38  REGEN_PURGE  "STATE Regen Hot Purge" %
%   N10:0  SYSTEM_STATE  "STATE The current state of the system" %
%   N9:0  SYSTEM_STANDBY  "STATE System Standby" %
%   N13:3  REGEN_STANDBY_BUFFER  "state The state when the system went to SYSTEM STANDBY" %
%   N9:29  REGEN_IDLE %
% Rung: 31 %
% REGEN PURGE
% If the state of this machine is REGEN PURGE, run a timer and counter to measure the elapsed minutes of regen run. %
SOR EQU N13:0 N9:38 BST XIO T4:56/DN TON T4:56 1.0 60 0 NXB XIC T4:56/DN CTU C5:8 480 0 BND EOR
%   N13:0  REGEN_STATE  "STATE The current state of the regen process" %
%   N9:38  REGEN_PURGE  "STATE Regen Hot Purge" %
%   T4:56  REGEN_PURGE_SEC_TMR  "TIMER Regen purge (seconds)" %
%   C5:8  REGEN_PURGE_MINUTES  "COUNTER Regen THe number of minutes the purge step runs" %
% Rung: 32 %
SOR LEQ N7:14 300 EQU N13:0 N9:38 GEQ C5:8.ACC 5 LEQ C5:8.ACC 35 BST XIO T4:94/DN TON T4:94 1.0 90 0 NXB LEQ T4:94.ACC 59 OTE B34:1/0 BND EOR
%   N7:14  PURIFIER_SIZE %
%   N13:0  REGEN_STATE  "STATE The current state of the regen process" %
%   N9:38  REGEN_PURGE  "STATE Regen Hot Purge" %
%   C5:8  REGEN_PURGE_MINUTES  "COUNTER Regen THe number of minutes the purge step runs" %
%   T4:94  CYCLE_PURGE_TMR %
%   B34:1/0  AV11_CYCLE_PURGE %
% Rung: 33 %
SOR LEQ N7:14 300 GRT C5:8.ACC 35 OTU B34:1/0 EOR
%   N7:14  PURIFIER_SIZE %
%   C5:8  REGEN_PURGE_MINUTES  "COUNTER Regen THe number of minutes the purge step runs" %
%   B34:1/0  AV11_CYCLE_PURGE %

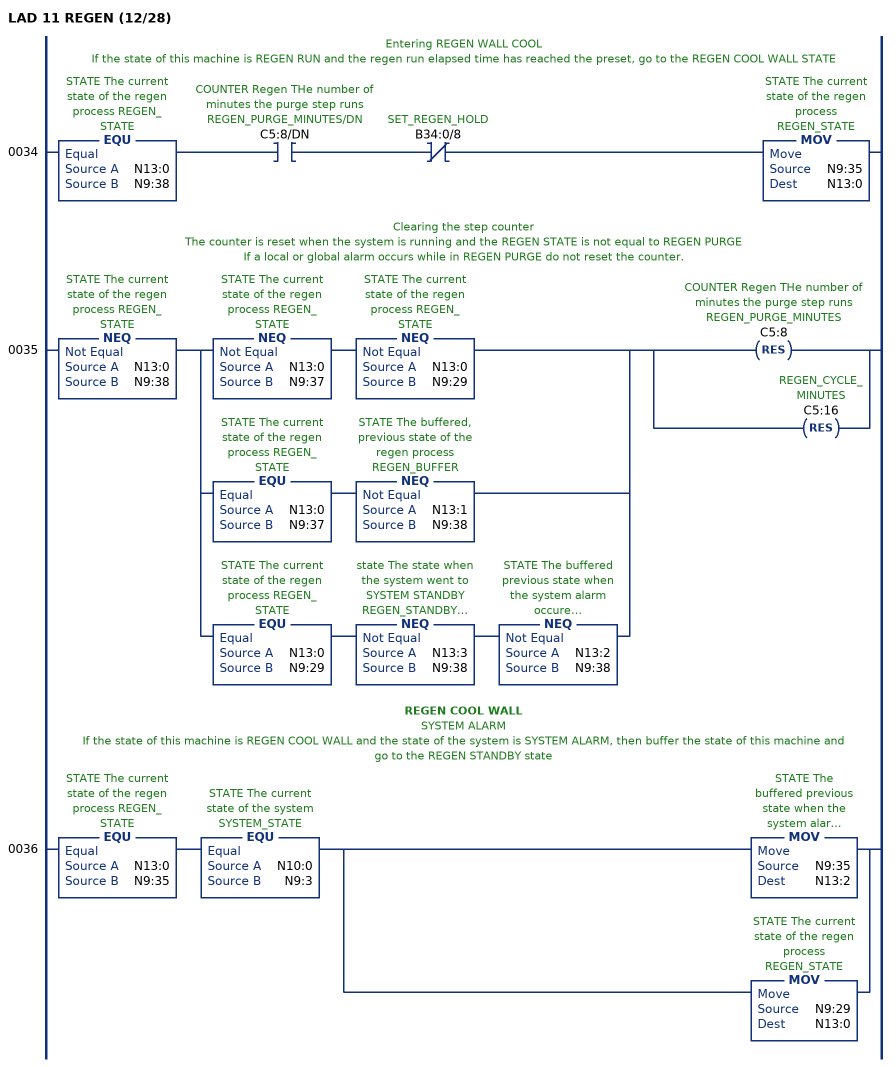
% Rung: 34 %
% Entering REGEN WALL COOL
% If the state of this machine is REGEN RUN and the regen run elapsed time has reached the preset, go to the REGEN COOL WALL STATE %
SOR EQU N13:0 N9:38 XIC C5:8/DN XIO B34:0/8 MOV N9:35 N13:0 EOR
%   N13:0  REGEN_STATE  "STATE The current state of the regen process" %
%   N9:38  REGEN_PURGE  "STATE Regen Hot Purge" %
%   C5:8  REGEN_PURGE_MINUTES  "COUNTER Regen THe number of minutes the purge step runs" %
%   B34:0/8  SET_REGEN_HOLD %
%   N9:35  REGEN_COOL_WALL  "STATE Regen Cool wall" %
% Rung: 35 %
% Clearing the step counter
% The counter is reset when the system is running and the REGEN STATE is not equal to REGEN PURGE
% If a local or global alarm occurs while in REGEN PURGE do not reset the counter. %
SOR NEQ N13:0 N9:38 BST NEQ N13:0 N9:37 NEQ N13:0 N9:29 NXB EQU N13:0 N9:37 NEQ N13:1 N9:38 NXB EQU N13:0 N9:29 NEQ N13:3 N9:38 NEQ N13:2 N9:38 BND BST RES C5:8 NXB RES C5:16 BND EOR
%   N13:0  REGEN_STATE  "STATE The current state of the regen process" %
%   N9:38  REGEN_PURGE  "STATE Regen Hot Purge" %
%   N9:37  REGEN_ALARM  "STATE Regen Alarm" %
%   N9:29  REGEN_IDLE %
%   N13:1  REGEN_BUFFER  "STATE The buffered, previous state of the regen process" %
%   N13:3  REGEN_STANDBY_BUFFER  "state The state when the system went to SYSTEM STANDBY" %
%   N13:2  REGEN_ALARM_BUFFER  "STATE The buffered previous state when the system alarm occured" %
%   C5:8  REGEN_PURGE_MINUTES  "COUNTER Regen THe number of minutes the purge step runs" %
%   C5:16  REGEN_CYCLE_MINUTES %
% Rung: 36 %
% TITLE: REGEN COOL WALL %
% SYSTEM ALARM
% If the state of this machine is REGEN COOL WALL and the state of the system is SYSTEM ALARM, then buffer the state of this machine and go to the REGEN STANDBY state %
SOR EQU N13:0 N9:35 EQU N10:0 N9:3 BST MOV N9:35 N13:2 NXB MOV N9:29 N13:0 BND EOR
%   N13:0  REGEN_STATE  "STATE The current state of the regen process" %
%   N9:35  REGEN_COOL_WALL  "STATE Regen Cool wall" %
%   N10:0  SYSTEM_STATE  "STATE The current state of the system" %
%   N9:3  SYSTEM_ALARM  "STATE System Alarm" %
%   N13:2  REGEN_ALARM_BUFFER  "STATE The buffered previous state when the system alarm occured" %
%   N9:29  REGEN_IDLE %

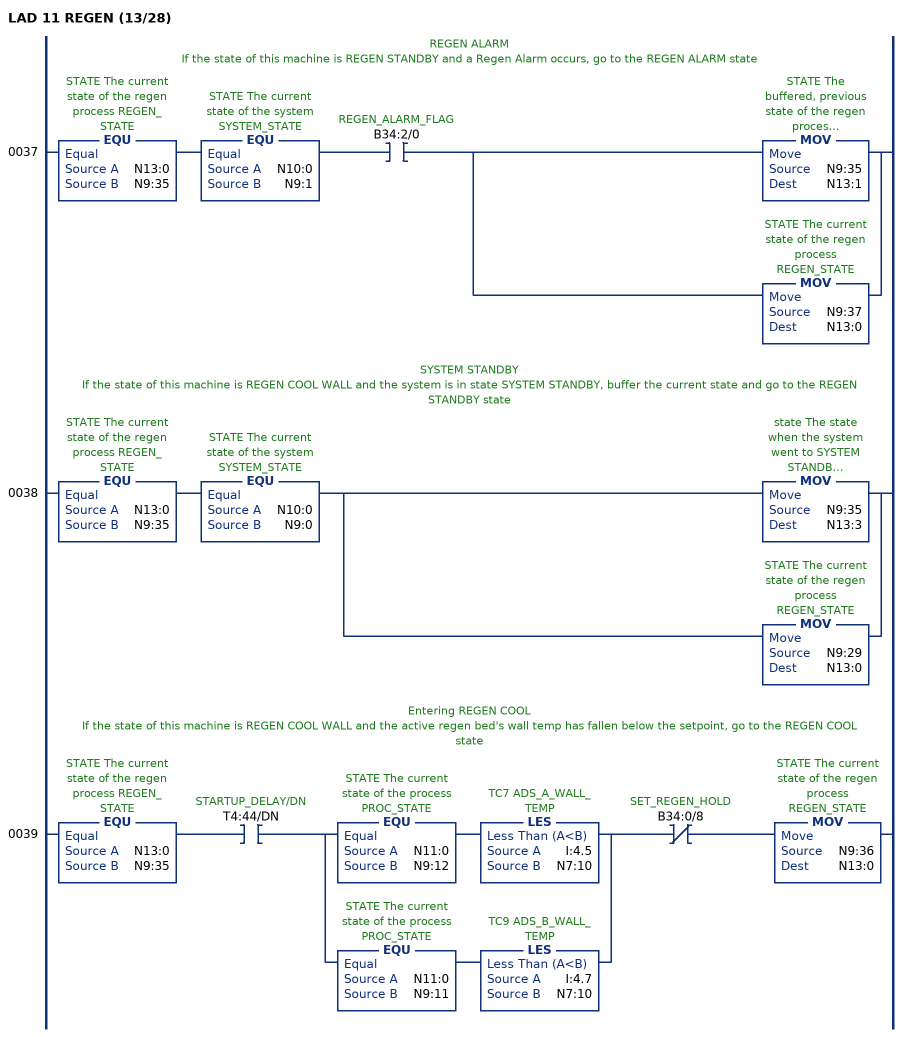
% Rung: 37 %
% REGEN ALARM
% If the state of this machine is REGEN STANDBY and a Regen Alarm occurs, go to the REGEN ALARM state %
SOR EQU N13:0 N9:35 EQU N10:0 N9:1 XIC B34:2/0 BST MOV N9:35 N13:1 NXB MOV N9:37 N13:0 BND EOR
%   N13:0  REGEN_STATE  "STATE The current state of the regen process" %
%   N9:35  REGEN_COOL_WALL  "STATE Regen Cool wall" %
%   N10:0  SYSTEM_STATE  "STATE The current state of the system" %
%   N9:1  SYSTEM_PROCESS  "STATE System Process" %
%   B34:2/0  REGEN_ALARM_FLAG %
%   N13:1  REGEN_BUFFER  "STATE The buffered, previous state of the regen process" %
%   N9:37  REGEN_ALARM  "STATE Regen Alarm" %
% Rung: 38 %
% SYSTEM STANDBY
% If the state of this machine is REGEN COOL WALL and the system is in state SYSTEM STANDBY, buffer the current state and go to the REGEN STANDBY state %
SOR EQU N13:0 N9:35 EQU N10:0 N9:0 BST MOV N9:35 N13:3 NXB MOV N9:29 N13:0 BND EOR
%   N13:0  REGEN_STATE  "STATE The current state of the regen process" %
%   N9:35  REGEN_COOL_WALL  "STATE Regen Cool wall" %
%   N10:0  SYSTEM_STATE  "STATE The current state of the system" %
%   N9:0  SYSTEM_STANDBY  "STATE System Standby" %
%   N13:3  REGEN_STANDBY_BUFFER  "state The state when the system went to SYSTEM STANDBY" %
%   N9:29  REGEN_IDLE %
% Rung: 39 %
% Entering REGEN COOL
% If the state of this machine is REGEN COOL WALL and the active regen bed's wall temp has fallen below the setpoint, go to the REGEN COOL state %
SOR EQU N13:0 N9:35 XIC T4:44/DN BST EQU N11:0 N9:12 LES I:4.5 N7:10 NXB EQU N11:0 N9:11 LES I:4.7 N7:10 BND XIO B34:0/8 MOV N9:36 N13:0 EOR
%   N13:0  REGEN_STATE  "STATE The current state of the regen process" %
%   N9:35  REGEN_COOL_WALL  "STATE Regen Cool wall" %
%   T4:44  STARTUP_DELAY %
%   N11:0  PROC_STATE  "STATE The current state of the process" %
%   N9:12  PROC_PURIFY_B  "STATE Process Purify B" %
%   I:4.5  ADS_A_WALL_TEMP  "TC7" %
%   N7:10  ADS_WALL_TEMP_COOL  "CONFIG The temp at which the adsorber wall is deemed to be cool enough to purify" %
%   N9:11  PROC_PURIFY_A  "STATE Process Purify A" %
%   I:4.7  ADS_B_WALL_TEMP  "TC9" %
%   B34:0/8  SET_REGEN_HOLD %
%   N9:36  REGEN_COOL  "STATE Regen Cool" %

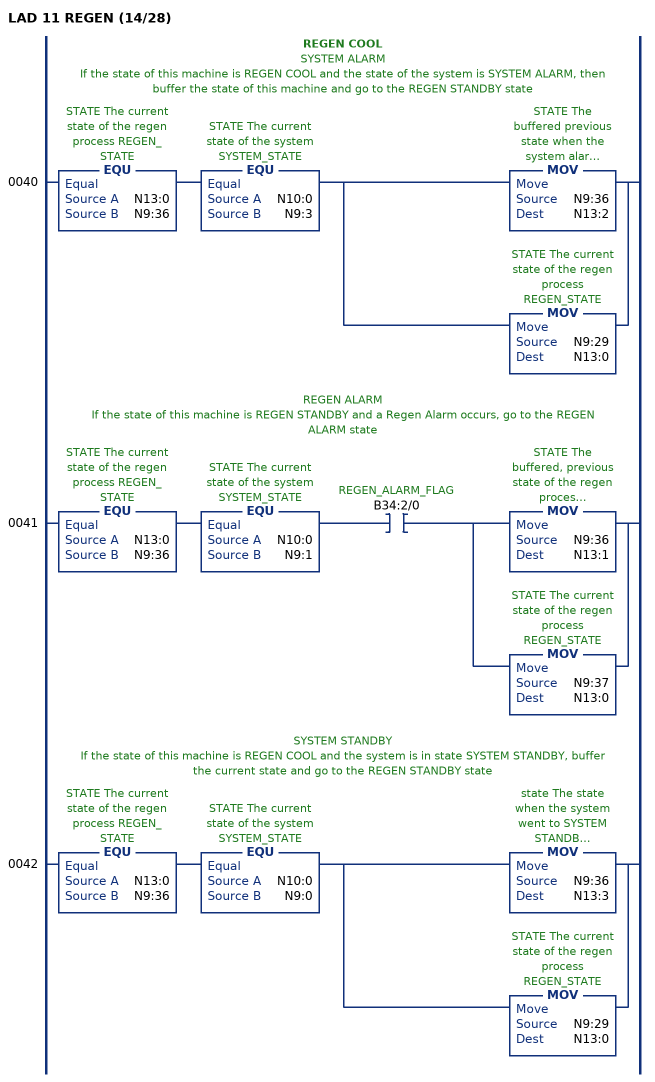
% Rung: 40 %
% TITLE: REGEN COOL %
% SYSTEM ALARM
% If the state of this machine is REGEN COOL and the state of the system is SYSTEM ALARM, then buffer the state of this machine and go to the REGEN STANDBY state %
SOR EQU N13:0 N9:36 EQU N10:0 N9:3 BST MOV N9:36 N13:2 NXB MOV N9:29 N13:0 BND EOR
%   N13:0  REGEN_STATE  "STATE The current state of the regen process" %
%   N9:36  REGEN_COOL  "STATE Regen Cool" %
%   N10:0  SYSTEM_STATE  "STATE The current state of the system" %
%   N9:3  SYSTEM_ALARM  "STATE System Alarm" %
%   N13:2  REGEN_ALARM_BUFFER  "STATE The buffered previous state when the system alarm occured" %
%   N9:29  REGEN_IDLE %
% Rung: 41 %
% REGEN ALARM
% If the state of this machine is REGEN STANDBY and a Regen Alarm occurs, go to the REGEN ALARM state %
SOR EQU N13:0 N9:36 EQU N10:0 N9:1 XIC B34:2/0 BST MOV N9:36 N13:1 NXB MOV N9:37 N13:0 BND EOR
%   N13:0  REGEN_STATE  "STATE The current state of the regen process" %
%   N9:36  REGEN_COOL  "STATE Regen Cool" %
%   N10:0  SYSTEM_STATE  "STATE The current state of the system" %
%   N9:1  SYSTEM_PROCESS  "STATE System Process" %
%   B34:2/0  REGEN_ALARM_FLAG %
%   N13:1  REGEN_BUFFER  "STATE The buffered, previous state of the regen process" %
%   N9:37  REGEN_ALARM  "STATE Regen Alarm" %
% Rung: 42 %
% SYSTEM STANDBY
% If the state of this machine is REGEN COOL and the system is in state SYSTEM STANDBY, buffer the current state and go to the REGEN STANDBY state %
SOR EQU N13:0 N9:36 EQU N10:0 N9:0 BST MOV N9:36 N13:3 NXB MOV N9:29 N13:0 BND EOR
%   N13:0  REGEN_STATE  "STATE The current state of the regen process" %
%   N9:36  REGEN_COOL  "STATE Regen Cool" %
%   N10:0  SYSTEM_STATE  "STATE The current state of the system" %
%   N9:0  SYSTEM_STANDBY  "STATE System Standby" %
%   N13:3  REGEN_STANDBY_BUFFER  "state The state when the system went to SYSTEM STANDBY" %
%   N9:29  REGEN_IDLE %

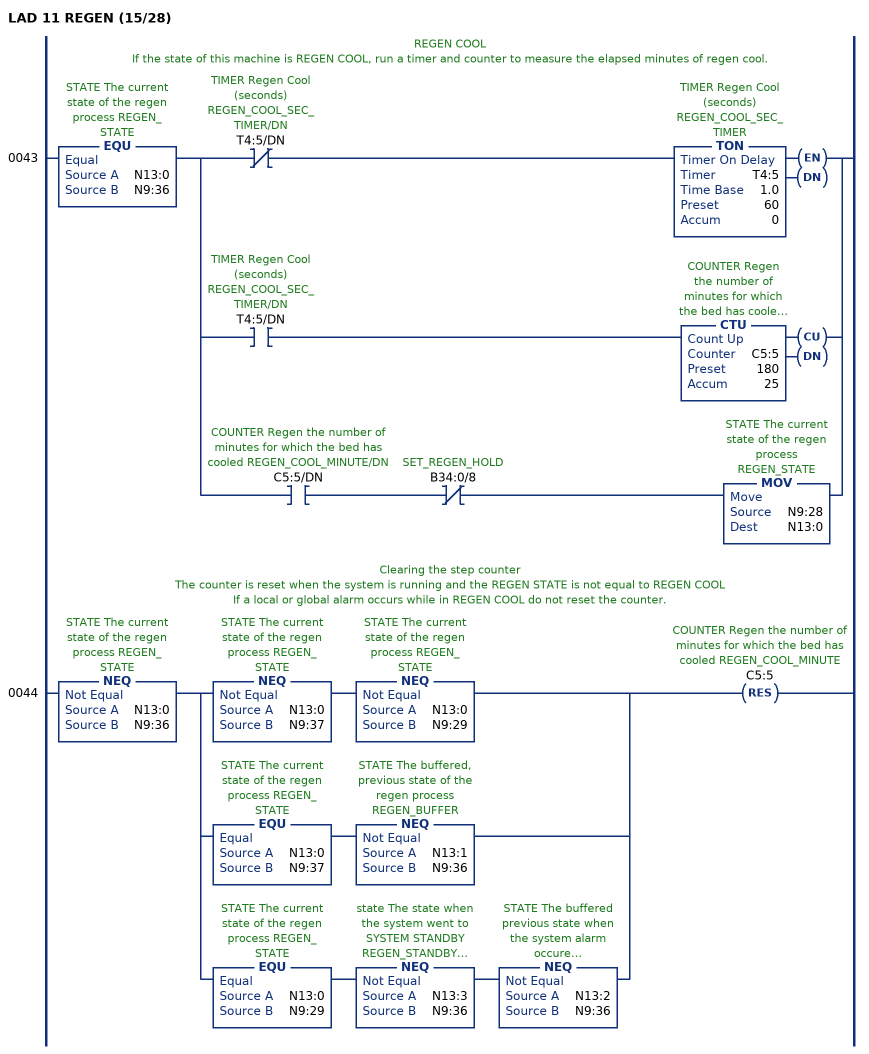
% Rung: 43 %
% REGEN COOL
% If the state of this machine is REGEN COOL, run a timer and counter to measure the elapsed minutes of regen cool. %
SOR EQU N13:0 N9:36 BST XIO T4:5/DN TON T4:5 1.0 60 0 NXB XIC T4:5/DN CTU C5:5 180 25 NXB XIC C5:5/DN XIO B34:0/8 MOV N9:28 N13:0 BND EOR
%   N13:0  REGEN_STATE  "STATE The current state of the regen process" %
%   N9:36  REGEN_COOL  "STATE Regen Cool" %
%   T4:5  REGEN_COOL_SEC_TIMER  "TIMER Regen Cool (seconds)" %
%   C5:5  REGEN_COOL_MINUTE  "COUNTER Regen the number of minutes for which the bed has cooled" %
%   B34:0/8  SET_REGEN_HOLD %
%   N9:28  REGEN_VENT_2  "STATE Regen Vent 2" %
% Rung: 44 %
% Clearing the step counter
% The counter is reset when the system is running and the REGEN STATE is not equal to REGEN COOL
% If a local or global alarm occurs while in REGEN COOL do not reset the counter. %
SOR NEQ N13:0 N9:36 BST NEQ N13:0 N9:37 NEQ N13:0 N9:29 NXB EQU N13:0 N9:37 NEQ N13:1 N9:36 NXB EQU N13:0 N9:29 NEQ N13:3 N9:36 NEQ N13:2 N9:36 BND RES C5:5 EOR
%   N13:0  REGEN_STATE  "STATE The current state of the regen process" %
%   N9:36  REGEN_COOL  "STATE Regen Cool" %
%   N9:37  REGEN_ALARM  "STATE Regen Alarm" %
%   N9:29  REGEN_IDLE %
%   N13:1  REGEN_BUFFER  "STATE The buffered, previous state of the regen process" %
%   N13:3  REGEN_STANDBY_BUFFER  "state The state when the system went to SYSTEM STANDBY" %
%   N13:2  REGEN_ALARM_BUFFER  "STATE The buffered previous state when the system alarm occured" %
%   C5:5  REGEN_COOL_MINUTE  "COUNTER Regen the number of minutes for which the bed has cooled" %

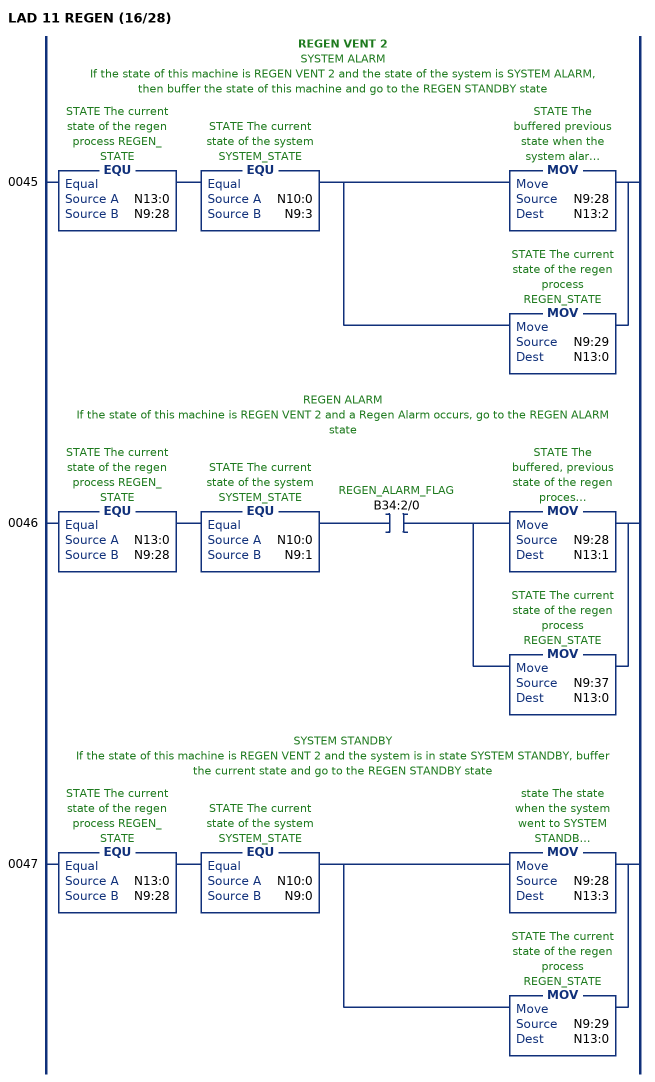
% Rung: 45 %
% TITLE: REGEN VENT 2 %
% SYSTEM ALARM
% If the state of this machine is REGEN VENT 2 and the state of the system is SYSTEM ALARM, then buffer the state of this machine and go to the REGEN STANDBY state %
SOR EQU N13:0 N9:28 EQU N10:0 N9:3 BST MOV N9:28 N13:2 NXB MOV N9:29 N13:0 BND EOR
%   N13:0  REGEN_STATE  "STATE The current state of the regen process" %
%   N9:28  REGEN_VENT_2  "STATE Regen Vent 2" %
%   N10:0  SYSTEM_STATE  "STATE The current state of the system" %
%   N9:3  SYSTEM_ALARM  "STATE System Alarm" %
%   N13:2  REGEN_ALARM_BUFFER  "STATE The buffered previous state when the system alarm occured" %
%   N9:29  REGEN_IDLE %
% Rung: 46 %
% REGEN ALARM
% If the state of this machine is REGEN VENT 2 and a Regen Alarm occurs, go to the REGEN ALARM state %
SOR EQU N13:0 N9:28 EQU N10:0 N9:1 XIC B34:2/0 BST MOV N9:28 N13:1 NXB MOV N9:37 N13:0 BND EOR
%   N13:0  REGEN_STATE  "STATE The current state of the regen process" %
%   N9:28  REGEN_VENT_2  "STATE Regen Vent 2" %
%   N10:0  SYSTEM_STATE  "STATE The current state of the system" %
%   N9:1  SYSTEM_PROCESS  "STATE System Process" %
%   B34:2/0  REGEN_ALARM_FLAG %
%   N13:1  REGEN_BUFFER  "STATE The buffered, previous state of the regen process" %
%   N9:37  REGEN_ALARM  "STATE Regen Alarm" %
% Rung: 47 %
% SYSTEM STANDBY
% If the state of this machine is REGEN VENT 2 and the system is in state SYSTEM STANDBY, buffer the current state and go to the REGEN STANDBY state %
SOR EQU N13:0 N9:28 EQU N10:0 N9:0 BST MOV N9:28 N13:3 NXB MOV N9:29 N13:0 BND EOR
%   N13:0  REGEN_STATE  "STATE The current state of the regen process" %
%   N9:28  REGEN_VENT_2  "STATE Regen Vent 2" %
%   N10:0  SYSTEM_STATE  "STATE The current state of the system" %
%   N9:0  SYSTEM_STANDBY  "STATE System Standby" %
%   N13:3  REGEN_STANDBY_BUFFER  "state The state when the system went to SYSTEM STANDBY" %
%   N9:29  REGEN_IDLE %

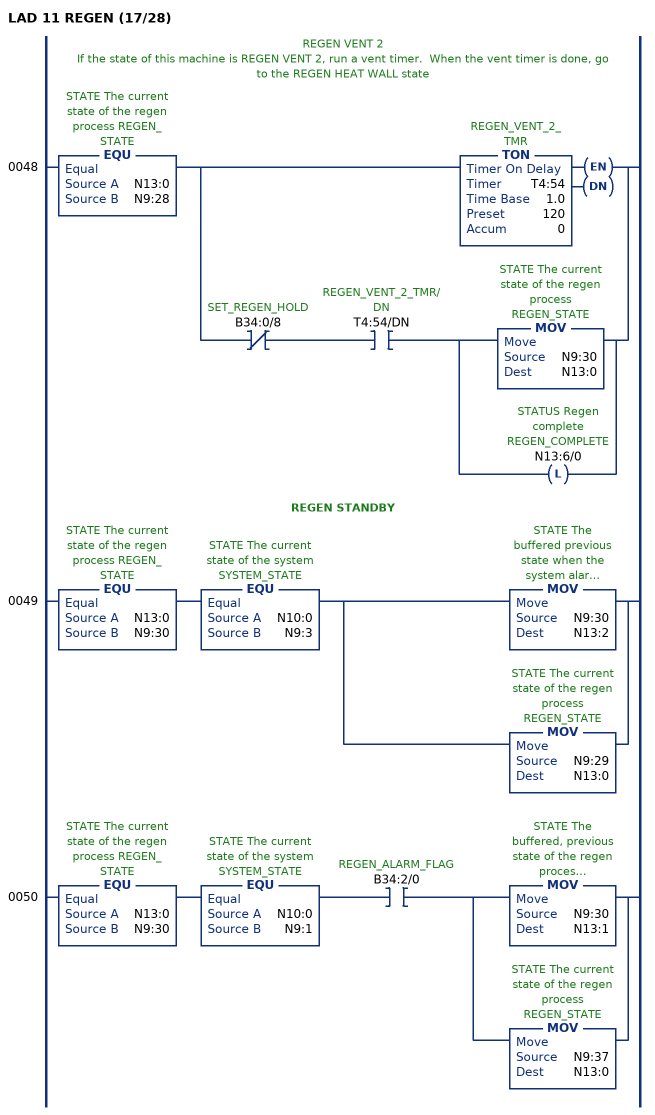
% Rung: 48 %
% REGEN VENT 2
% If the state of this machine is REGEN VENT 2, run a vent timer.  When the vent timer is done, go to the REGEN HEAT WALL state %
SOR EQU N13:0 N9:28 BST TON T4:54 1.0 120 0 NXB XIO B34:0/8 XIC T4:54/DN BST MOV N9:30 N13:0 NXB OTL N13:6/0 BND BND EOR
%   N13:0  REGEN_STATE  "STATE The current state of the regen process" %
%   N9:28  REGEN_VENT_2  "STATE Regen Vent 2" %
%   T4:54  REGEN_VENT_2_TMR %
%   B34:0/8  SET_REGEN_HOLD %
%   N9:30  REGEN_STANDBY  "STATE Regen Standby" %
%   N13:6/0  REGEN_COMPLETE  "STATUS Regen complete" %
% Rung: 49 %
% TITLE: REGEN STANDBY %
SOR EQU N13:0 N9:30 EQU N10:0 N9:3 BST MOV N9:30 N13:2 NXB MOV N9:29 N13:0 BND EOR
%   N13:0  REGEN_STATE  "STATE The current state of the regen process" %
%   N9:30  REGEN_STANDBY  "STATE Regen Standby" %
%   N10:0  SYSTEM_STATE  "STATE The current state of the system" %
%   N9:3  SYSTEM_ALARM  "STATE System Alarm" %
%   N13:2  REGEN_ALARM_BUFFER  "STATE The buffered previous state when the system alarm occured" %
%   N9:29  REGEN_IDLE %
% Rung: 50 %
SOR EQU N13:0 N9:30 EQU N10:0 N9:1 XIC B34:2/0 BST MOV N9:30 N13:1 NXB MOV N9:37 N13:0 BND EOR
%   N13:0  REGEN_STATE  "STATE The current state of the regen process" %
%   N9:30  REGEN_STANDBY  "STATE Regen Standby" %
%   N10:0  SYSTEM_STATE  "STATE The current state of the system" %
%   N9:1  SYSTEM_PROCESS  "STATE System Process" %
%   B34:2/0  REGEN_ALARM_FLAG %
%   N13:1  REGEN_BUFFER  "STATE The buffered, previous state of the regen process" %
%   N9:37  REGEN_ALARM  "STATE Regen Alarm" %

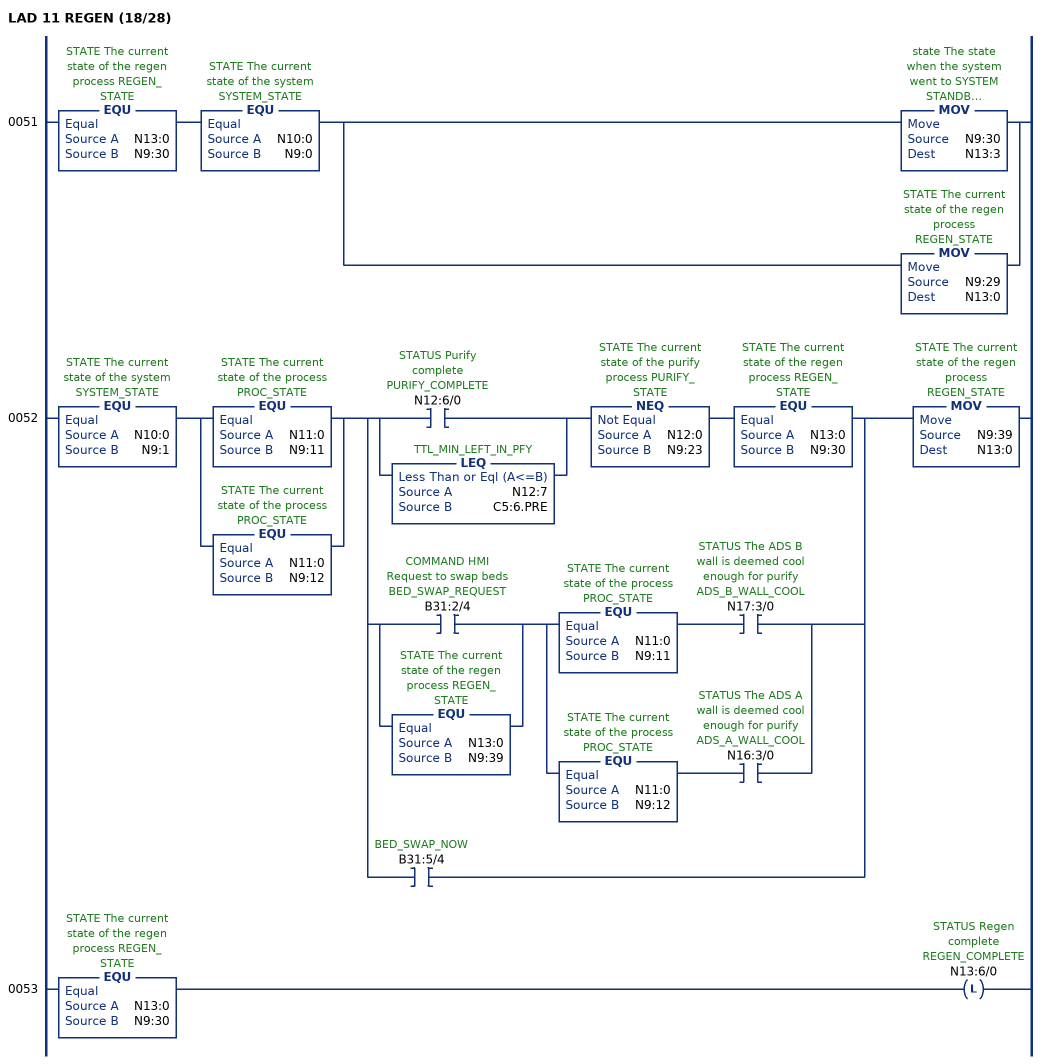
% Rung: 51 %
SOR EQU N13:0 N9:30 EQU N10:0 N9:0 BST MOV N9:30 N13:3 NXB MOV N9:29 N13:0 BND EOR
%   N13:0  REGEN_STATE  "STATE The current state of the regen process" %
%   N9:30  REGEN_STANDBY  "STATE Regen Standby" %
%   N10:0  SYSTEM_STATE  "STATE The current state of the system" %
%   N9:0  SYSTEM_STANDBY  "STATE System Standby" %
%   N13:3  REGEN_STANDBY_BUFFER  "state The state when the system went to SYSTEM STANDBY" %
%   N9:29  REGEN_IDLE %
% Rung: 52 %
SOR EQU N10:0 N9:1 BST EQU N11:0 N9:11 NXB EQU N11:0 N9:12 BND BST BST XIC N12:6/0 NXB LEQ N12:7 C5:6.PRE BND NEQ N12:0 N9:23 EQU N13:0 N9:30 NXB BST XIC B31:2/4 NXB EQU N13:0 N9:39 BND BST EQU N11:0 N9:11 XIC N17:3/0 NXB EQU N11:0 N9:12 XIC N16:3/0 BND NXB XIC B31:5/4 BND MOV N9:39 N13:0 EOR
%   N10:0  SYSTEM_STATE  "STATE The current state of the system" %
%   N9:1  SYSTEM_PROCESS  "STATE System Process" %
%   N11:0  PROC_STATE  "STATE The current state of the process" %
%   N9:11  PROC_PURIFY_A  "STATE Process Purify A" %
%   N9:12  PROC_PURIFY_B  "STATE Process Purify B" %
%   N12:6/0  PURIFY_COMPLETE  "STATUS Purify complete" %
%   N12:7  TTL_MIN_LEFT_IN_PFY %
%   C5:6  REGEN_EQUALIZE_MIN %
%   N12:0  PURIFY_STATE  "STATE The current state of the purify process" %
%   N9:23  PURIFY_MANUAL_HOLD  "STATE Purify Manual Hold" %
%   N13:0  REGEN_STATE  "STATE The current state of the regen process" %
%   N9:30  REGEN_STANDBY  "STATE Regen Standby" %
%   B31:2/4  BED_SWAP_REQUEST  "COMMAND HMI Request to swap beds" %
%   N9:39  REGEN_EQUALIZE %
%   N17:3/0  ADS_B_WALL_COOL  "STATUS The ADS B wall is deemed cool enough for purify" %
%   N16:3/0  ADS_A_WALL_COOL  "STATUS The ADS A wall is deemed cool enough for purify" %
%   B31:5/4  BED_SWAP_NOW %
% Rung: 53 %
SOR EQU N13:0 N9:30 OTL N13:6/0 EOR
%   N13:0  REGEN_STATE  "STATE The current state of the regen process" %
%   N9:30  REGEN_STANDBY  "STATE Regen Standby" %
%   N13:6/0  REGEN_COMPLETE  "STATUS Regen complete" %

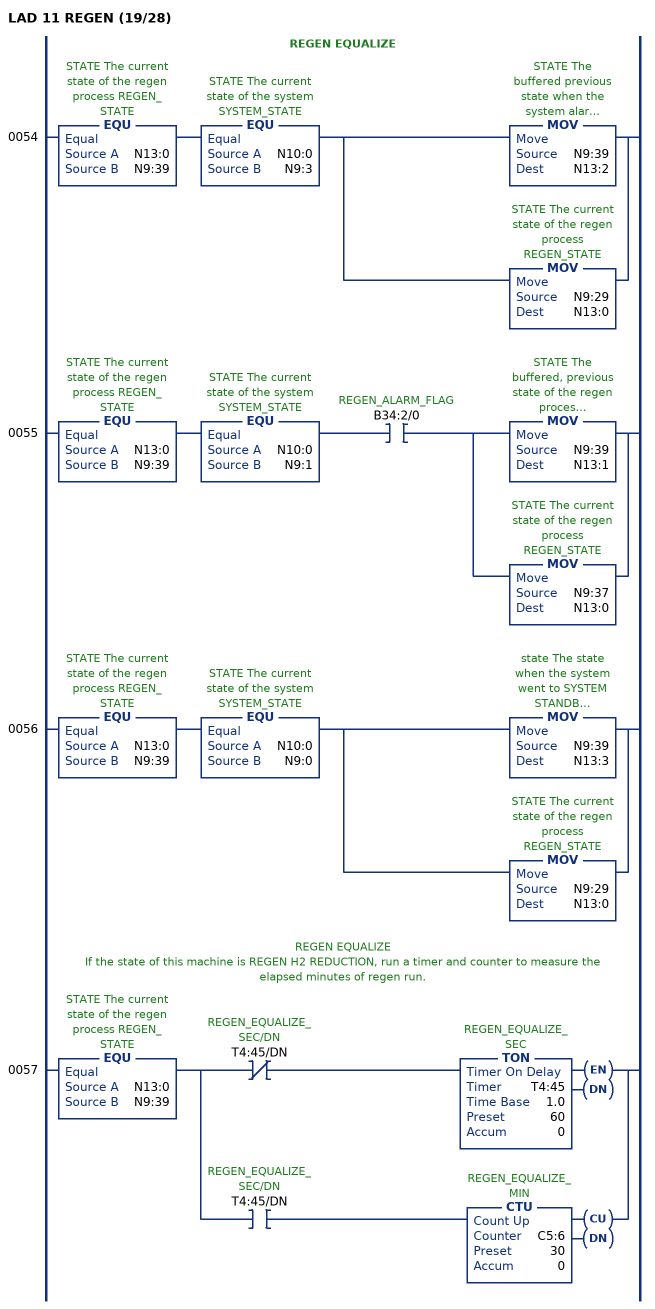
% Rung: 54 %
% TITLE: REGEN EQUALIZE %
SOR EQU N13:0 N9:39 EQU N10:0 N9:3 BST MOV N9:39 N13:2 NXB MOV N9:29 N13:0 BND EOR
%   N13:0  REGEN_STATE  "STATE The current state of the regen process" %
%   N9:39  REGEN_EQUALIZE %
%   N10:0  SYSTEM_STATE  "STATE The current state of the system" %
%   N9:3  SYSTEM_ALARM  "STATE System Alarm" %
%   N13:2  REGEN_ALARM_BUFFER  "STATE The buffered previous state when the system alarm occured" %
%   N9:29  REGEN_IDLE %
% Rung: 55 %
SOR EQU N13:0 N9:39 EQU N10:0 N9:1 XIC B34:2/0 BST MOV N9:39 N13:1 NXB MOV N9:37 N13:0 BND EOR
%   N13:0  REGEN_STATE  "STATE The current state of the regen process" %
%   N9:39  REGEN_EQUALIZE %
%   N10:0  SYSTEM_STATE  "STATE The current state of the system" %
%   N9:1  SYSTEM_PROCESS  "STATE System Process" %
%   B34:2/0  REGEN_ALARM_FLAG %
%   N13:1  REGEN_BUFFER  "STATE The buffered, previous state of the regen process" %
%   N9:37  REGEN_ALARM  "STATE Regen Alarm" %
% Rung: 56 %
SOR EQU N13:0 N9:39 EQU N10:0 N9:0 BST MOV N9:39 N13:3 NXB MOV N9:29 N13:0 BND EOR
%   N13:0  REGEN_STATE  "STATE The current state of the regen process" %
%   N9:39  REGEN_EQUALIZE %
%   N10:0  SYSTEM_STATE  "STATE The current state of the system" %
%   N9:0  SYSTEM_STANDBY  "STATE System Standby" %
%   N13:3  REGEN_STANDBY_BUFFER  "state The state when the system went to SYSTEM STANDBY" %
%   N9:29  REGEN_IDLE %
% Rung: 57 %
% REGEN EQUALIZE
% If the state of this machine is REGEN H2 REDUCTION, run a timer and counter to measure the elapsed minutes of regen run. %
SOR EQU N13:0 N9:39 BST XIO T4:45/DN TON T4:45 1.0 60 0 NXB XIC T4:45/DN CTU C5:6 30 0 BND EOR
%   N13:0  REGEN_STATE  "STATE The current state of the regen process" %
%   N9:39  REGEN_EQUALIZE %
%   T4:45  REGEN_EQUALIZE_SEC %
%   C5:6  REGEN_EQUALIZE_MIN %

